LIN {X 0,Y 370.907,Z 638.749,A -85,B 0,C 180,E1 -12853.488,E2 -12853.488} C_VEL
LIN {X 0,Y 369.621,Z 646.813,A -85,B 0,C 180,E1 -12855.864,E2 -12855.864} C_VEL
LIN {X 0,Y 368.614,Z 653.844,A -85,B 0,C 180,E1 -12858.452,E2 -12858.452} C_VEL
LIN {X 0,Y 367.975,Z 659.585,A -85,B 0,C 180,E1 -12861.211,E2 -12861.211} C_VEL
LIN {X 0,Y 367.683,Z 663.304,A -85,B 0,C 180,E1 -12863.69,E2 -12863.69} C_VEL
LIN {X 0,Y 367.515,Z 665.39,A -85,B 0,C 180,E1 -12865.613,E2 -12865.613} C_VEL
LIN {X 0,Y 367.433,Z 666.778,A -85,B 0,C 180,E1 -12867.808,E2 -12867.808} C_VEL
LIN {X 0,Y 367.455,Z 667.313,A -85,B 0,C 180,E1 -12870,E2 -12870} C_VEL
LIN {X 0,Y 367.425,Z 666.872,A -85,B 0,C 180,E1 -12872.034,E2 -12872.034} C_VEL
LIN {X 0,Y 366.804,Z 666.517,A -85,B 0,C 180,E1 -12872.948,E2 -12872.948} C_VEL
LIN {X 0,Y 364.039,Z 665.625,A -85,B 0,C 180,E1 -12874.433,E2 -12874.433} C_VEL
LIN {X 0,Y 361.697,Z 664.56,A -85,B 0,C 180,E1 -12875.627,E2 -12875.627} C_VEL
LIN {X 0,Y 360.71,Z 663.504,A -85,B 0,C 180,E1 -12876.542,E2 -12876.542} C_VEL
LIN {X 0,Y 360.64,Z 663.097,A -85,B 0,C 180,E1 -12876.85,E2 -12876.85} C_VEL
LIN {X 0,Y 361.004,Z 658.926,A -85,B 0,C 180,E1 -12879.525,E2 -12879.525} C_VEL
LIN {X 0,Y 361.59,Z 654.287,A -85,B 0,C 180,E1 -12881.776,E2 -12881.776} C_VEL
LIN {X 0,Y 362.727,Z 646.801,A -85,B 0,C 180,E1 -12884.589,E2 -12884.589} C_VEL
LIN {X 0,Y 364.17,Z 638.314,A -85,B 0,C 180,E1 -12887.116,E2 -12887.116} C_VEL
LIN {X 0,Y 365.899,Z 628.97,A -85,B 0,C 180,E1 -12889.392,E2 -12889.392} C_VEL
LIN {X 0,Y 367.605,Z 619.716,A -85,B 0,C 180,E1 -12891.3,E2 -12891.3} C_VEL
LIN {X 0,Y 369.724,Z 608.71,A -85,B 0,C 180,E1 -12893.23,E2 -12893.23} C_VEL
LIN {X 0,Y 372.107,Z 596.049,A -85,B 0,C 180,E1 -12895.093,E2 -12895.093} C_VEL
LIN {X 0,Y 374.536,Z 582.365,A -85,B 0,C 180,E1 -12896.766,E2 -12896.766} C_VEL
LIN {X 0,Y 376.71,Z 569.237,A -85,B 0,C 180,E1 -12898.103,E2 -12898.103} C_VEL
LIN {X 0,Y 378.659,Z 555.105,A -85,B 0,C 180,E1 -12899.324,E2 -12899.324} C_VEL
LIN {X 0,Y 380.626,Z 540.226,A -85,B 0,C 180,E1 -12900.362,E2 -12900.362} C_VEL
LIN {X 0,Y 382.44,Z 523.413,A -85,B 0,C 180,E1 -12901.274,E2 -12901.274} C_VEL
LIN {X 0,Y 383.681,Z 507.284,A -85,B 0,C 180,E1 -12901.932,E2 -12901.932} C_VEL
LIN {X 0,Y 384.653,Z 490.648,A -85,B 0,C 180,E1 -12902.392,E2 -12902.392} C_VEL
LIN {X 0,Y 389.159,Z 339.278,A -85,B 0,C 180,E1 -12905.281,E2 -12905.281} C_VEL
LIN {X 0,Y 378.091,Z 317.354,A -85,B 0,C 180,E1 -12906.995,E2 -12906.995} C_VEL
LIN {X 0,Y 369.152,Z 301.874,A -85,B 0,C 180,E1 -12908.431,E2 -12908.431} C_VEL
LIN {X 0,Y 364.671,Z 294.925,A -85,B 0,C 180,E1 -12909.169,E2 -12909.169} C_VEL
LIN {X 0,Y 362.414,Z 291.756,A -85,B 0,C 180,E1 -12909.542,E2 -12909.542} C_VEL
LIN {X 0,Y 361.846,Z 289.718,A -85,B 0,C 180,E1 -12909.687,E2 -12909.687} C_VEL
LIN {X 0,Y 361.835,Z 289.718,A -85,B 0,C 180,E1 -12912.828,E2 -12912.828} C_VEL
LIN {X 0,Y 361.816,Z 289.719,A -85,B 0,C 180,E1 -12915.946,E2 -12915.946} C_VEL
LIN {X 0,Y 361.833,Z 289.715,A -85,B 0,C 180,E1 -12919.244,E2 -12919.244} C_VEL
LIN {X 0,Y 361.861,Z 289.71,A -85,B 0,C 180,E1 -12922.777,E2 -12922.777} C_VEL
LIN {X 0,Y 361.852,Z 289.721,A -85,B 0,C 180,E1 -12925.719,E2 -12925.719} C_VEL
LIN {X 0,Y 361.871,Z 289.722,A -85,B 0,C 180,E1 -12929.672,E2 -12929.672} C_VEL
LIN {X 0,Y 361.952,Z 289.699,A -85,B 0,C 180,E1 -12933.475,E2 -12933.475} C_VEL
LIN {X 0,Y 361.889,Z 289.7,A -85,B 0,C 180,E1 -12937.144,E2 -12937.144} C_VEL
LIN {X 0,Y 361.906,Z 289.717,A -85,B 0,C 180,E1 -12940.723,E2 -12940.723} C_VEL
LIN {X 0,Y 361.93,Z 289.693,A -85,B 0,C 180,E1 -12943.066,E2 -12943.066} C_VEL
LIN {X 0,Y 361.996,Z 289.703,A -85,B 0,C 180,E1 -12946.528,E2 -12946.528} C_VEL
LIN {X 0,Y 362.029,Z 289.677,A -85,B 0,C 180,E1 -12949.938,E2 -12949.938} C_VEL
LIN {X 0,Y 362.149,Z 289.678,A -85,B 0,C 180,E1 -12952.192,E2 -12952.192} C_VEL
LIN {X 0,Y 362.116,Z 289.69,A -85,B 0,C 180,E1 -12954.431,E2 -12954.431} C_VEL
LIN {X 0,Y 362.278,Z 289.647,A -85,B 0,C 180,E1 -12957.776,E2 -12957.776} C_VEL
LIN {X 0,Y 362.425,Z 289.65,A -85,B 0,C 180,E1 -12960,E2 -12960} C_VEL
LIN {X 0,Y 362.28,Z 289.662,A -85,B 0,C 180,E1 -12962.223,E2 -12962.223} C_VEL
LIN {X 0,Y 362.17,Z 289.682,A -85,B 0,C 180,E1 -12966.686,E2 -12966.686} C_VEL
LIN {X 0,Y 362.071,Z 289.684,A -85,B 0,C 180,E1 -12968.933,E2 -12968.933} C_VEL
LIN {X 0,Y 361.957,Z 289.702,A -85,B 0,C 180,E1 -12972.332,E2 -12972.332} C_VEL
LIN {X 0,Y 361.959,Z 289.709,A -85,B 0,C 180,E1 -12974.62,E2 -12974.62} C_VEL
LIN {X 0,Y 361.957,Z 289.707,A -85,B 0,C 180,E1 -12978.099,E2 -12978.099} C_VEL
LIN {X 0,Y 361.889,Z 289.717,A -85,B 0,C 180,E1 -12981.653,E2 -12981.653} C_VEL
LIN {X 0,Y 361.925,Z 289.718,A -85,B 0,C 180,E1 -12985.29,E2 -12985.29} C_VEL
LIN {X 0,Y 361.915,Z 289.716,A -85,B 0,C 180,E1 -12987.778,E2 -12987.778} C_VEL
LIN {X 0,Y 361.844,Z 289.731,A -85,B 0,C 180,E1 -12991.285,E2 -12991.285} C_VEL
LIN {X 0,Y 361.851,Z 289.729,A -85,B 0,C 180,E1 -12994.28,E2 -12994.28} C_VEL
LIN {X 0,Y 361.862,Z 289.728,A -85,B 0,C 180,E1 -12997.223,E2 -12997.223} C_VEL
LIN {X 0,Y 361.833,Z 289.733,A -85,B 0,C 180,E1 -13000.756,E2 -13000.756} C_VEL
LIN {X 0,Y 361.816,Z 289.734,A -85,B 0,C 180,E1 -13004.368,E2 -13004.368} C_VEL
LIN {X 0,Y 361.831,Z 289.732,A -85,B 0,C 180,E1 -13007.744,E2 -13007.744} C_VEL
LIN {X 0,Y 366.657,Z 302.939,A -85,B 0,C 180,E1 -13010.56,E2 -13010.56} C_VEL
LIN {X 0,Y 367.781,Z 306.002,A -85,B 0,C 180,E1 -13011.134,E2 -13011.134} C_VEL
LIN {X 0,Y 378.049,Z 324.644,A -85,B 0,C 180,E1 -13012.805,E2 -13012.805} C_VEL
LIN {X 0,Y 387.494,Z 344.135,A -85,B 0,C 180,E1 -13014.286,E2 -13014.286} C_VEL
LIN {X 0,Y 388.307,Z 346.732,A -85,B 0,C 180,E1 -13014.43,E2 -13014.43} C_VEL
LIN {X 0,Y 388.915,Z 352.418,A -85,B 0,C 180,E1 -13014.619,E2 -13014.619} C_VEL
LIN {X 0,Y 384.083,Z 512.924,A -85,B 0,C 180,E1 -13017.685,E2 -13017.685} C_VEL
LIN {X 0,Y 382.968,Z 528.887,A -85,B 0,C 180,E1 -13018.157,E2 -13018.157} C_VEL
LIN {X 0,Y 381.501,Z 544.325,A -85,B 0,C 180,E1 -13018.794,E2 -13018.794} C_VEL
LIN {X 0,Y 379.765,Z 559.811,A -85,B 0,C 180,E1 -13019.639,E2 -13019.639} C_VEL
LIN {X 0,Y 377.615,Z 575.779,A -85,B 0,C 180,E1 -13020.755,E2 -13020.755} C_VEL
LIN {X 0,Y 375.218,Z 591.049,A -85,B 0,C 180,E1 -13022.079,E2 -13022.079} C_VEL
LIN {X 0,Y 372.743,Z 605.042,A -85,B 0,C 180,E1 -13023.549,E2 -13023.549} C_VEL
LIN {X 0,Y 370.628,Z 617.005,A -85,B 0,C 180,E1 -13025.045,E2 -13025.045} C_VEL
LIN {X 0,Y 368.639,Z 628.246,A -85,B 0,C 180,E1 -13026.697,E2 -13026.697} C_VEL
LIN {X 0,Y 366.551,Z 639.457,A -85,B 0,C 180,E1 -13028.636,E2 -13028.636} C_VEL
LIN {X 0,Y 364.551,Z 650.326,A -85,B 0,C 180,E1 -13030.869,E2 -13030.869} C_VEL
LIN {X 0,Y 363.096,Z 659.472,A -85,B 0,C 180,E1 -13033.122,E2 -13033.122} C_VEL
LIN {X 0,Y 361.974,Z 667.139,A -85,B 0,C 180,E1 -13035.38,E2 -13035.38} C_VEL
LIN {X 0,Y 361.197,Z 673.403,A -85,B 0,C 180,E1 -13037.641,E2 -13037.641} C_VEL
LIN {X 0,Y 360.634,Z 678.538,A -85,B 0,C 180,E1 -13039.899,E2 -13039.899} C_VEL
LIN {X 0,Y 360.451,Z 682.536,A -85,B 0,C 180,E1 -13042.156,E2 -13042.156} C_VEL
LIN {X 0,Y 360.326,Z 685.494,A -85,B 0,C 180,E1 -13044.404,E2 -13044.404} C_VEL
LIN {X 0,Y 360.277,Z 687.443,A -85,B 0,C 180,E1 -13046.645,E2 -13046.645} C_VEL
LIN {X 0,Y 360.312,Z 688.409,A -85,B 0,C 180,E1 -13048.882,E2 -13048.882} C_VEL
LIN {X 0,Y 360.312,Z 688.408,A -85,B 0,C 180,E1 -13051.118,E2 -13051.118} C_VEL
LIN {X 0,Y 360.277,Z 687.435,A -85,B 0,C 180,E1 -13053.355,E2 -13053.355} C_VEL
LIN {X 0,Y 360.375,Z 685.105,A -85,B 0,C 180,E1 -13055.962,E2 -13055.962} C_VEL
LIN {X 0,Y 360.451,Z 682.522,A -85,B 0,C 180,E1 -13057.844,E2 -13057.844} C_VEL
LIN {X 0,Y 360.634,Z 678.523,A -85,B 0,C 180,E1 -13060.101,E2 -13060.101} C_VEL
LIN {X 0,Y 361.194,Z 673.38,A -85,B 0,C 180,E1 -13062.359,E2 -13062.359} C_VEL
LIN {X 0,Y 361.973,Z 667.108,A -85,B 0,C 180,E1 -13064.62,E2 -13064.62} C_VEL
LIN {X 0,Y 363.295,Z 658.416,A -85,B 0,C 180,E1 -13067.158,E2 -13067.158} C_VEL
LIN {X 0,Y 364.819,Z 649.165,A -85,B 0,C 180,E1 -13069.379,E2 -13069.379} C_VEL
LIN {X 0,Y 366.566,Z 639.399,A -85,B 0,C 180,E1 -13071.363,E2 -13071.363} C_VEL
LIN {X 0,Y 368.709,Z 628.173,A -85,B 0,C 180,E1 -13073.298,E2 -13073.298} C_VEL
LIN {X 0,Y 370.837,Z 615.941,A -85,B 0,C 180,E1 -13075.09,E2 -13075.09} C_VEL
LIN {X 0,Y 373.179,Z 602.583,A -85,B 0,C 180,E1 -13076.72,E2 -13076.72} C_VEL
LIN {X 0,Y 375.461,Z 589.361,A -85,B 0,C 180,E1 -13078.067,E2 -13078.067} C_VEL
LIN {X 0,Y 377.374,Z 577.294,A -85,B 0,C 180,E1 -13079.113,E2 -13079.113} C_VEL
LIN {X 0,Y 379.367,Z 562.609,A -85,B 0,C 180,E1 -13080.166,E2 -13080.166} C_VEL
LIN {X 0,Y 381.26,Z 546.692,A -85,B 0,C 180,E1 -13081.074,E2 -13081.074} C_VEL
LIN {X 0,Y 382.736,Z 531.3,A -85,B 0,C 180,E1 -13081.749,E2 -13081.749} C_VEL
LIN {X 0,Y 384.045,Z 514.1,A -85,B 0,C 180,E1 -13082.273,E2 -13082.273} C_VEL
LIN {X 0,Y 388.906,Z 351.926,A -85,B 0,C 180,E1 -13085.377,E2 -13085.377} C_VEL
LIN {X 0,Y 388.013,Z 345.342,A -85,B 0,C 180,E1 -13085.616,E2 -13085.616} C_VEL
LIN {X 0,Y 379.342,Z 327.267,A -85,B 0,C 180,E1 -13086.969,E2 -13086.969} C_VEL
LIN {X 0,Y 369.961,Z 309.878,A -85,B 0,C 180,E1 -13088.481,E2 -13088.481} C_VEL
LIN {X 0,Y 367.493,Z 305.339,A -85,B 0,C 180,E1 -13088.93,E2 -13088.93} C_VEL
LIN {X 0,Y 363.709,Z 294.968,A -85,B 0,C 180,E1 -13091.097,E2 -13091.097} C_VEL
LIN {X 0,Y 361.832,Z 289.724,A -85,B 0,C 180,E1 -13092.271,E2 -13092.271} C_VEL
LIN {X 0,Y 361.833,Z 289.72,A -85,B 0,C 180,E1 -13095.944,E2 -13095.944} C_VEL
LIN {X 0,Y 361.833,Z 289.724,A -85,B 0,C 180,E1 -13099.245,E2 -13099.245} C_VEL
LIN {X 0,Y 361.861,Z 289.715,A -85,B 0,C 180,E1 -13102.777,E2 -13102.777} C_VEL
LIN {X 0,Y 361.852,Z 289.721,A -85,B 0,C 180,E1 -13105.72,E2 -13105.72} C_VEL
LIN {X 0,Y 361.872,Z 289.716,A -85,B 0,C 180,E1 -13109.672,E2 -13109.672} C_VEL
LIN {X 0,Y 361.952,Z 289.711,A -85,B 0,C 180,E1 -13113.475,E2 -13113.475} C_VEL
LIN {X 0,Y 361.89,Z 289.721,A -85,B 0,C 180,E1 -13117.145,E2 -13117.145} C_VEL
LIN {X 0,Y 361.909,Z 289.693,A -85,B 0,C 180,E1 -13120.724,E2 -13120.724} C_VEL
LIN {X 0,Y 361.931,Z 289.716,A -85,B 0,C 180,E1 -13123.066,E2 -13123.066} C_VEL
LIN {X 0,Y 361.996,Z 289.677,A -85,B 0,C 180,E1 -13126.528,E2 -13126.528} C_VEL
LIN {X 0,Y 362.029,Z 289.701,A -85,B 0,C 180,E1 -13129.938,E2 -13129.938} C_VEL
LIN {X 0,Y 362.161,Z 289.655,A -85,B 0,C 180,E1 -13133.314,E2 -13133.314} C_VEL
LIN {X 0,Y 362.281,Z 289.668,A -85,B 0,C 180,E1 -13137.777,E2 -13137.777} C_VEL
LIN {X 0,Y 362.424,Z 289.626,A -85,B 0,C 180,E1 -13140,E2 -13140} C_VEL
LIN {X 0,Y 362.279,Z 289.653,A -85,B 0,C 180,E1 -13142.224,E2 -13142.224} C_VEL
LIN {X 0,Y 362.161,Z 289.665,A -85,B 0,C 180,E1 -13146.687,E2 -13146.687} C_VEL
LIN {X 0,Y 362.03,Z 289.692,A -85,B 0,C 180,E1 -13150.062,E2 -13150.062} C_VEL
LIN {X 0,Y 361.996,Z 289.69,A -85,B 0,C 180,E1 -13153.899,E2 -13153.899} C_VEL
LIN {X 0,Y 361.966,Z 289.707,A -85,B 0,C 180,E1 -13157.939,E2 -13157.939} C_VEL
LIN {X 0,Y 361.882,Z 289.692,A -85,B 0,C 180,E1 -13161.654,E2 -13161.654} C_VEL
LIN {X 0,Y 361.927,Z 289.714,A -85,B 0,C 180,E1 -13165.29,E2 -13165.29} C_VEL
LIN {X 0,Y 361.907,Z 289.692,A -85,B 0,C 180,E1 -13167.779,E2 -13167.779} C_VEL
LIN {X 0,Y 361.836,Z 289.72,A -85,B 0,C 180,E1 -13171.63,E2 -13171.63} C_VEL
LIN {X 0,Y 361.873,Z 289.72,A -85,B 0,C 180,E1 -13175.345,E2 -13175.345} C_VEL
LIN {X 0,Y 361.867,Z 289.707,A -85,B 0,C 180,E1 -13179.027,E2 -13179.027} C_VEL
LIN {X 0,Y 361.835,Z 289.711,A -85,B 0,C 180,E1 -13182.829,E2 -13182.829} C_VEL
LIN {X 0,Y 361.816,Z 289.715,A -85,B 0,C 180,E1 -13185.947,E2 -13185.947} C_VEL
LIN {X 0,Y 361.835,Z 289.727,A -85,B 0,C 180,E1 -13189.245,E2 -13189.245} C_VEL
LIN {X 0,Y 361.839,Z 289.728,A -85,B 0,C 180,E1 -13190.441,E2 -13190.441} C_VEL
LIN {X 0,Y 362.896,Z 292.623,A -85,B 0,C 180,E1 -13190.657,E2 -13190.657} C_VEL
LIN {X 0,Y 364.71,Z 294.95,A -85,B 0,C 180,E1 -13190.95,E2 -13190.95} C_VEL
LIN {X 0,Y 372.447,Z 307.404,A -85,B 0,C 180,E1 -13192.216,E2 -13192.216} C_VEL
LIN {X 0,Y 380.406,Z 321.844,A -85,B 0,C 180,E1 -13193.481,E2 -13193.481} C_VEL
LIN {X 0,Y 389.033,Z 339.103,A -85,B 0,C 180,E1 -13194.808,E2 -13194.808} C_VEL
LIN {X 0,Y 384.556,Z 492.624,A -85,B 0,C 180,E1 -13197.755,E2 -13197.755} C_VEL
LIN {X 0,Y 383.59,Z 508.462,A -85,B 0,C 180,E1 -13198.214,E2 -13198.214} C_VEL
LIN {X 0,Y 382.299,Z 524.246,A -85,B 0,C 180,E1 -13198.867,E2 -13198.867} C_VEL
LIN {X 0,Y 380.624,Z 539.824,A -85,B 0,C 180,E1 -13199.715,E2 -13199.715} C_VEL
LIN {X 0,Y 378.562,Z 555.625,A -85,B 0,C 180,E1 -13200.818,E2 -13200.818} C_VEL
LIN {X 0,Y 376.568,Z 569.681,A -85,B 0,C 180,E1 -13202.036,E2 -13202.036} C_VEL
LIN {X 0,Y 374.451,Z 582.728,A -85,B 0,C 180,E1 -13203.378,E2 -13203.378} C_VEL
LIN {X 0,Y 372.228,Z 595.02,A -85,B 0,C 180,E1 -13204.871,E2 -13204.871} C_VEL
LIN {X 0,Y 370.133,Z 606.325,A -85,B 0,C 180,E1 -13206.501,E2 -13206.501} C_VEL
LIN {X 0,Y 367.956,Z 617.73,A -85,B 0,C 180,E1 -13208.428,E2 -13208.428} C_VEL
LIN {X 0,Y 366.253,Z 626.909,A -85,B 0,C 180,E1 -13210.251,E2 -13210.251} C_VEL
LIN {X 0,Y 364.597,Z 635.754,A -85,B 0,C 180,E1 -13212.326,E2 -13212.326} C_VEL
LIN {X 0,Y 363.367,Z 642.912,A -85,B 0,C 180,E1 -13214.29,E2 -13214.29} C_VEL
LIN {X 0,Y 362.22,Z 649.717,A -85,B 0,C 180,E1 -13216.536,E2 -13216.536} C_VEL
LIN {X 0,Y 361.389,Z 655.303,A -85,B 0,C 180,E1 -13218.786,E2 -13218.786} C_VEL
LIN {X 0,Y 360.944,Z 659.793,A -85,B 0,C 180,E1 -13221.039,E2 -13221.039} C_VEL
LIN {X 0,Y 360.587,Z 663.718,A -85,B 0,C 180,E1 -13223.727,E2 -13223.727} C_VEL
LIN {X 0,Y 360.449,Z 665.597,A -85,B 0,C 180,E1 -13225.527,E2 -13225.527} C_VEL
LIN {X 0,Y 360.334,Z 666.986,A -85,B 0,C 180,E1 -13227.764,E2 -13227.764} C_VEL
LIN {X 0,Y 360.359,Z 667.52,A -85,B 0,C 180,E1 -13230,E2 -13230} C_VEL
LIN {X 0,Y 360.334,Z 667.029,A -85,B 0,C 180,E1 -13232.236,E2 -13232.236} C_VEL
LIN {X 0,Y 360.448,Z 665.682,A -85,B 0,C 180,E1 -13234.473,E2 -13234.473} C_VEL
LIN {X 0,Y 360.64,Z 663.097,A -85,B 0,C 180,E1 -13236.85,E2 -13236.85} C_VEL
LIN {X 0,Y 360.022,Z 661.911,A -85,B 0,C 180,E1 -13237.763,E2 -13237.763} C_VEL
LIN {X 0,Y 357.323,Z 659.723,A -85,B 0,C 180,E1 -13239.249,E2 -13239.249} C_VEL
LIN {X 0,Y 354.789,Z 657.157,A -85,B 0,C 180,E1 -13240.741,E2 -13240.741} C_VEL
LIN {X 0,Y 354.443,Z 655.273,A -85,B 0,C 180,E1 -13241.65,E2 -13241.65} C_VEL
LIN {X 0,Y 355.247,Z 650.204,A -85,B 0,C 180,E1 -13243.733,E2 -13243.733} C_VEL
LIN {X 0,Y 356.422,Z 643.435,A -85,B 0,C 180,E1 -13246.025,E2 -13246.025} C_VEL
LIN {X 0,Y 357.944,Z 635.243,A -85,B 0,C 180,E1 -13248.309,E2 -13248.309} C_VEL
LIN {X 0,Y 359.824,Z 625.486,A -85,B 0,C 180,E1 -13250.583,E2 -13250.583} C_VEL
LIN {X 0,Y 361.853,Z 615.447,A -85,B 0,C 180,E1 -13252.556,E2 -13252.556} C_VEL
LIN {X 0,Y 364.176,Z 603.608,A -85,B 0,C 180,E1 -13254.514,E2 -13254.514} C_VEL
LIN {X 0,Y 366.713,Z 590.572,A -85,B 0,C 180,E1 -13256.307,E2 -13256.307} C_VEL
LIN {X 0,Y 368.98,Z 577.552,A -85,B 0,C 180,E1 -13257.817,E2 -13257.817} C_VEL
LIN {X 0,Y 371.334,Z 563.556,A -85,B 0,C 180,E1 -13259.166,E2 -13259.166} C_VEL
LIN {X 0,Y 373.238,Z 550.201,A -85,B 0,C 180,E1 -13260.244,E2 -13260.244} C_VEL
LIN {X 0,Y 375.08,Z 535.938,A -85,B 0,C 180,E1 -13261.172,E2 -13261.172} C_VEL
LIN {X 0,Y 376.727,Z 519.187,A -85,B 0,C 180,E1 -13262.04,E2 -13262.04} C_VEL
LIN {X 0,Y 378.038,Z 503.614,A -85,B 0,C 180,E1 -13262.624,E2 -13262.624} C_VEL
LIN {X 0,Y 378.868,Z 486.851,A -85,B 0,C 180,E1 -13263.053,E2 -13263.053} C_VEL
LIN {X 0,Y 383.292,Z 341.409,A -85,B 0,C 180,E1 -13265.859,E2 -13265.859} C_VEL
LIN {X 0,Y 372.607,Z 320.441,A -85,B 0,C 180,E1 -13267.563,E2 -13267.563} C_VEL
LIN {X 0,Y 364.726,Z 306.671,A -85,B 0,C 180,E1 -13268.869,E2 -13268.869} C_VEL
LIN {X 0,Y 358.95,Z 298.084,A -85,B 0,C 180,E1 -13269.841,E2 -13269.841} C_VEL
LIN {X 0,Y 357.037,Z 294.944,A -85,B 0,C 180,E1 -13270.18,E2 -13270.18} C_VEL
LIN {X 0,Y 355.371,Z 292.659,A -85,B 0,C 180,E1 -13270.468,E2 -13270.468} C_VEL
LIN {X 0,Y 354.794,Z 290.6,A -85,B 0,C 180,E1 -13270.637,E2 -13270.637} C_VEL
LIN {X 0,Y 354.766,Z 290.608,A -85,B 0,C 180,E1 -13273.896,E2 -13273.896} C_VEL
LIN {X 0,Y 354.793,Z 290.601,A -85,B 0,C 180,E1 -13277.662,E2 -13277.662} C_VEL
LIN {X 0,Y 354.814,Z 290.6,A -85,B 0,C 180,E1 -13280.666,E2 -13280.666} C_VEL
LIN {X 0,Y 354.82,Z 290.596,A -85,B 0,C 180,E1 -13284.3,E2 -13284.3} C_VEL
LIN {X 0,Y 354.785,Z 290.588,A -85,B 0,C 180,E1 -13287.666,E2 -13287.666} C_VEL
LIN {X 0,Y 354.844,Z 290.58,A -85,B 0,C 180,E1 -13291.618,E2 -13291.618} C_VEL
LIN {X 0,Y 354.897,Z 290.587,A -85,B 0,C 180,E1 -13294.172,E2 -13294.172} C_VEL
LIN {X 0,Y 354.833,Z 290.574,A -85,B 0,C 180,E1 -13297.894,E2 -13297.894} C_VEL
LIN {X 0,Y 354.92,Z 290.582,A -85,B 0,C 180,E1 -13301.891,E2 -13301.891} C_VEL
LIN {X 0,Y 354.941,Z 290.58,A -85,B 0,C 180,E1 -13305.981,E2 -13305.981} C_VEL
LIN {X 0,Y 354.975,Z 290.557,A -85,B 0,C 180,E1 -13309.736,E2 -13309.736} C_VEL
LIN {X 0,Y 355.112,Z 290.552,A -85,B 0,C 180,E1 -13312.037,E2 -13312.037} C_VEL
LIN {X 0,Y 355.09,Z 290.565,A -85,B 0,C 180,E1 -13314.321,E2 -13314.321} C_VEL
LIN {X 0,Y 355.241,Z 290.522,A -85,B 0,C 180,E1 -13317.732,E2 -13317.732} C_VEL
LIN {X 0,Y 355.395,Z 290.526,A -85,B 0,C 180,E1 -13320,E2 -13320} C_VEL
LIN {X 0,Y 355.243,Z 290.536,A -85,B 0,C 180,E1 -13322.267,E2 -13322.267} C_VEL
LIN {X 0,Y 355.136,Z 290.559,A -85,B 0,C 180,E1 -13326.819,E2 -13326.819} C_VEL
LIN {X 0,Y 355.013,Z 290.561,A -85,B 0,C 180,E1 -13329.112,E2 -13329.112} C_VEL
LIN {X 0,Y 354.918,Z 290.58,A -85,B 0,C 180,E1 -13332.581,E2 -13332.581} C_VEL
LIN {X 0,Y 354.887,Z 290.589,A -85,B 0,C 180,E1 -13336.096,E2 -13336.096} C_VEL
LIN {X 0,Y 354.904,Z 290.585,A -85,B 0,C 180,E1 -13338.472,E2 -13338.472} C_VEL
LIN {X 0,Y 354.832,Z 290.597,A -85,B 0,C 180,E1 -13342.106,E2 -13342.106} C_VEL
LIN {X 0,Y 354.897,Z 290.593,A -85,B 0,C 180,E1 -13345.827,E2 -13345.827} C_VEL
LIN {X 0,Y 354.851,Z 290.596,A -85,B 0,C 180,E1 -13349.679,E2 -13349.679} C_VEL
LIN {X 0,Y 354.803,Z 290.606,A -85,B 0,C 180,E1 -13353.702,E2 -13353.702} C_VEL
LIN {X 0,Y 354.796,Z 290.606,A -85,B 0,C 180,E1 -13356.459,E2 -13356.459} C_VEL
LIN {X 0,Y 354.821,Z 290.605,A -85,B 0,C 180,E1 -13359.424,E2 -13359.424} C_VEL
LIN {X 0,Y 354.785,Z 290.61,A -85,B 0,C 180,E1 -13362.867,E2 -13362.867} C_VEL
LIN {X 0,Y 354.799,Z 290.69,A -85,B 0,C 180,E1 -13366.918,E2 -13366.918} C_VEL
LIN {X 0,Y 359.992,Z 304.716,A -85,B 0,C 180,E1 -13370.018,E2 -13370.018} C_VEL
LIN {X 0,Y 360.489,Z 305.861,A -85,B 0,C 180,E1 -13370.196,E2 -13370.196} C_VEL
LIN {X 0,Y 370.78,Z 324.284,A -85,B 0,C 180,E1 -13371.945,E2 -13371.945} C_VEL
LIN {X 0,Y 379.91,Z 342.544,A -85,B 0,C 180,E1 -13373.429,E2 -13373.429} C_VEL
LIN {X 0,Y 382.62,Z 348.545,A -85,B 0,C 180,E1 -13373.864,E2 -13373.864} C_VEL
LIN {X 0,Y 383.121,Z 353.621,A -85,B 0,C 180,E1 -13374.033,E2 -13374.033} C_VEL
LIN {X 0,Y 378.075,Z 513.451,A -85,B 0,C 180,E1 -13377.126,E2 -13377.126} C_VEL
LIN {X 0,Y 376.874,Z 529.607,A -85,B 0,C 180,E1 -13377.619,E2 -13377.619} C_VEL
LIN {X 0,Y 375.269,Z 545.427,A -85,B 0,C 180,E1 -13378.295,E2 -13378.295} C_VEL
LIN {X 0,Y 373.489,Z 560.605,A -85,B 0,C 180,E1 -13379.152,E2 -13379.152} C_VEL
LIN {X 0,Y 371.387,Z 575.575,A -85,B 0,C 180,E1 -13380.215,E2 -13380.215} C_VEL
LIN {X 0,Y 368.906,Z 590.844,A -85,B 0,C 180,E1 -13381.558,E2 -13381.558} C_VEL
LIN {X 0,Y 366.354,Z 604.837,A -85,B 0,C 180,E1 -13383.05,E2 -13383.05} C_VEL
LIN {X 0,Y 364.069,Z 616.796,A -85,B 0,C 180,E1 -13384.564,E2 -13384.564} C_VEL
LIN {X 0,Y 362.036,Z 628.038,A -85,B 0,C 180,E1 -13386.246,E2 -13386.246} C_VEL
LIN {X 0,Y 359.839,Z 639.248,A -85,B 0,C 180,E1 -13388.218,E2 -13388.218} C_VEL
LIN {X 0,Y 357.782,Z 650.118,A -85,B 0,C 180,E1 -13390.492,E2 -13390.492} C_VEL
LIN {X 0,Y 356.204,Z 659.263,A -85,B 0,C 180,E1 -13392.785,E2 -13392.785} C_VEL
LIN {X 0,Y 355.007,Z 666.93,A -85,B 0,C 180,E1 -13395.087,E2 -13395.087} C_VEL
LIN {X 0,Y 354.191,Z 673.194,A -85,B 0,C 180,E1 -13397.393,E2 -13397.393} C_VEL
LIN {X 0,Y 353.578,Z 678.329,A -85,B 0,C 180,E1 -13399.695,E2 -13399.695} C_VEL
LIN {X 0,Y 353.362,Z 682.328,A -85,B 0,C 180,E1 -13401.997,E2 -13401.997} C_VEL
LIN {X 0,Y 353.259,Z 685.287,A -85,B 0,C 180,E1 -13404.291,E2 -13404.291} C_VEL
LIN {X 0,Y 353.197,Z 687.236,A -85,B 0,C 180,E1 -13406.578,E2 -13406.578} C_VEL
LIN {X 0,Y 353.212,Z 688.202,A -85,B 0,C 180,E1 -13408.86,E2 -13408.86} C_VEL
LIN {X 0,Y 353.212,Z 688.2,A -85,B 0,C 180,E1 -13411.14,E2 -13411.14} C_VEL
LIN {X 0,Y 353.197,Z 687.228,A -85,B 0,C 180,E1 -13413.422,E2 -13413.422} C_VEL
LIN {X 0,Y 353.275,Z 685.077,A -85,B 0,C 180,E1 -13415.908,E2 -13415.908} C_VEL
LIN {X 0,Y 353.362,Z 682.313,A -85,B 0,C 180,E1 -13418.003,E2 -13418.003} C_VEL
LIN {X 0,Y 353.578,Z 678.313,A -85,B 0,C 180,E1 -13420.305,E2 -13420.305} C_VEL
LIN {X 0,Y 354.188,Z 673.17,A -85,B 0,C 180,E1 -13422.607,E2 -13422.607} C_VEL
LIN {X 0,Y 355.006,Z 666.896,A -85,B 0,C 180,E1 -13424.913,E2 -13424.913} C_VEL
LIN {X 0,Y 356.431,Z 658.205,A -85,B 0,C 180,E1 -13427.499,E2 -13427.499} C_VEL
LIN {X 0,Y 358.026,Z 648.827,A -85,B 0,C 180,E1 -13429.792,E2 -13429.792} C_VEL
LIN {X 0,Y 359.848,Z 639.186,A -85,B 0,C 180,E1 -13431.782,E2 -13431.782} C_VEL
LIN {X 0,Y 362.085,Z 627.96,A -85,B 0,C 180,E1 -13433.75,E2 -13433.75} C_VEL
LIN {X 0,Y 364.317,Z 615.728,A -85,B 0,C 180,E1 -13435.571,E2 -13435.571} C_VEL
LIN {X 0,Y 366.789,Z 602.371,A -85,B 0,C 180,E1 -13437.224,E2 -13437.224} C_VEL
LIN {X 0,Y 369.299,Z 588.05,A -85,B 0,C 180,E1 -13438.697,E2 -13438.697} C_VEL
LIN {X 0,Y 371.621,Z 573.626,A -85,B 0,C 180,E1 -13439.92,E2 -13439.92} C_VEL
LIN {X 0,Y 373.773,Z 558.304,A -85,B 0,C 180,E1 -13440.979,E2 -13440.979} C_VEL
LIN {X 0,Y 375.571,Z 542.568,A -85,B 0,C 180,E1 -13441.834,E2 -13441.834} C_VEL
LIN {X 0,Y 377.076,Z 526.494,A -85,B 0,C 180,E1 -13442.48,E2 -13442.48} C_VEL
LIN {X 0,Y 378.261,Z 510.347,A -85,B 0,C 180,E1 -13442.922,E2 -13442.922} C_VEL
LIN {X 0,Y 383.037,Z 351.609,A -85,B 0,C 180,E1 -13446.004,E2 -13446.004} C_VEL
LIN {X 0,Y 382.42,Z 348.085,A -85,B 0,C 180,E1 -13446.151,E2 -13446.151} C_VEL
LIN {X 0,Y 373.879,Z 330.341,A -85,B 0,C 180,E1 -13447.524,E2 -13447.524} C_VEL
LIN {X 0,Y 365.281,Z 314.342,A -85,B 0,C 180,E1 -13448.952,E2 -13448.952} C_VEL
LIN {X 0,Y 360.178,Z 305.201,A -85,B 0,C 180,E1 -13449.854,E2 -13449.854} C_VEL
LIN {X 0,Y 355.516,Z 292.944,A -85,B 0,C 180,E1 -13452.556,E2 -13452.556} C_VEL
LIN {X 0,Y 354.782,Z 290.602,A -85,B 0,C 180,E1 -13453.079,E2 -13453.079} C_VEL
LIN {X 0,Y 354.778,Z 290.598,A -85,B 0,C 180,E1 -13456.106,E2 -13456.106} C_VEL
LIN {X 0,Y 354.785,Z 290.601,A -85,B 0,C 180,E1 -13459.179,E2 -13459.179} C_VEL
LIN {X 0,Y 354.804,Z 290.594,A -85,B 0,C 180,E1 -13462.403,E2 -13462.403} C_VEL
LIN {X 0,Y 354.809,Z 290.594,A -85,B 0,C 180,E1 -13464.941,E2 -13464.941} C_VEL
LIN {X 0,Y 354.791,Z 290.6,A -85,B 0,C 180,E1 -13468.405,E2 -13468.405} C_VEL
LIN {X 0,Y 354.849,Z 290.595,A -85,B 0,C 180,E1 -13471.619,E2 -13471.619} C_VEL
LIN {X 0,Y 354.897,Z 290.589,A -85,B 0,C 180,E1 -13474.173,E2 -13474.173} C_VEL
LIN {X 0,Y 354.834,Z 290.593,A -85,B 0,C 180,E1 -13477.894,E2 -13477.894} C_VEL
LIN {X 0,Y 354.92,Z 290.581,A -85,B 0,C 180,E1 -13481.892,E2 -13481.892} C_VEL
LIN {X 0,Y 354.94,Z 290.557,A -85,B 0,C 180,E1 -13485.981,E2 -13485.981} C_VEL
LIN {X 0,Y 354.976,Z 290.58,A -85,B 0,C 180,E1 -13489.736,E2 -13489.736} C_VEL
LIN {X 0,Y 355.124,Z 290.531,A -85,B 0,C 180,E1 -13493.181,E2 -13493.181} C_VEL
LIN {X 0,Y 355.244,Z 290.544,A -85,B 0,C 180,E1 -13497.733,E2 -13497.733} C_VEL
LIN {X 0,Y 355.373,Z 290.503,A -85,B 0,C 180,E1 -13500,E2 -13500} C_VEL
LIN {X 0,Y 355.242,Z 290.529,A -85,B 0,C 180,E1 -13502.268,E2 -13502.268} C_VEL
LIN {X 0,Y 355.124,Z 290.539,A -85,B 0,C 180,E1 -13506.82,E2 -13506.82} C_VEL
LIN {X 0,Y 354.976,Z 290.571,A -85,B 0,C 180,E1 -13510.264,E2 -13510.264} C_VEL
LIN {X 0,Y 354.941,Z 290.565,A -85,B 0,C 180,E1 -13514.019,E2 -13514.019} C_VEL
LIN {X 0,Y 354.921,Z 290.585,A -85,B 0,C 180,E1 -13518.109,E2 -13518.109} C_VEL
LIN {X 0,Y 354.829,Z 290.57,A -85,B 0,C 180,E1 -13522.107,E2 -13522.107} C_VEL
LIN {X 0,Y 354.898,Z 290.587,A -85,B 0,C 180,E1 -13525.828,E2 -13525.828} C_VEL
LIN {X 0,Y 354.845,Z 290.593,A -85,B 0,C 180,E1 -13529.68,E2 -13529.68} C_VEL
LIN {X 0,Y 354.805,Z 290.599,A -85,B 0,C 180,E1 -13533.702,E2 -13533.702} C_VEL
LIN {X 0,Y 354.797,Z 290.597,A -85,B 0,C 180,E1 -13536.46,E2 -13536.46} C_VEL
LIN {X 0,Y 354.823,Z 290.59,A -85,B 0,C 180,E1 -13539.424,E2 -13539.424} C_VEL
LIN {X 0,Y 354.787,Z 290.589,A -85,B 0,C 180,E1 -13542.867,E2 -13542.867} C_VEL
LIN {X 0,Y 354.765,Z 290.593,A -85,B 0,C 180,E1 -13546.104,E2 -13546.104} C_VEL
LIN {X 0,Y 354.789,Z 290.604,A -85,B 0,C 180,E1 -13549.503,E2 -13549.503} C_VEL
LIN {X 0,Y 355.805,Z 293.453,A -85,B 0,C 180,E1 -13549.728,E2 -13549.728} C_VEL
LIN {X 0,Y 357.773,Z 295.999,A -85,B 0,C 180,E1 -13550.063,E2 -13550.063} C_VEL
LIN {X 0,Y 359.906,Z 299.245,A -85,B 0,C 180,E1 -13550.431,E2 -13550.431} C_VEL
LIN {X 0,Y 367.872,Z 311.995,A -85,B 0,C 180,E1 -13551.769,E2 -13551.769} C_VEL
LIN {X 0,Y 375.815,Z 326.553,A -85,B 0,C 180,E1 -13553.068,E2 -13553.068} C_VEL
LIN {X 0,Y 383.232,Z 341.44,A -85,B 0,C 180,E1 -13554.242,E2 -13554.242} C_VEL
LIN {X 0,Y 378.542,Z 494.115,A -85,B 0,C 180,E1 -13557.212,E2 -13557.212} C_VEL
LIN {X 0,Y 377.432,Z 510.511,A -85,B 0,C 180,E1 -13557.712,E2 -13557.712} C_VEL
LIN {X 0,Y 375.997,Z 527.053,A -85,B 0,C 180,E1 -13558.442,E2 -13558.442} C_VEL
LIN {X 0,Y 374.126,Z 543.058,A -85,B 0,C 180,E1 -13559.367,E2 -13559.367} C_VEL
LIN {X 0,Y 372.049,Z 558.335,A -85,B 0,C 180,E1 -13560.486,E2 -13560.486} C_VEL
LIN {X 0,Y 369.818,Z 572.735,A -85,B 0,C 180,E1 -13561.789,E2 -13561.789} C_VEL
LIN {X 0,Y 367.401,Z 586.442,A -85,B 0,C 180,E1 -13563.287,E2 -13563.287} C_VEL
LIN {X 0,Y 365.031,Z 599.117,A -85,B 0,C 180,E1 -13564.94,E2 -13564.94} C_VEL
LIN {X 0,Y 362.944,Z 610.043,A -85,B 0,C 180,E1 -13566.612,E2 -13566.612} C_VEL
LIN {X 0,Y 360.701,Z 620.889,A -85,B 0,C 180,E1 -13568.572,E2 -13568.572} C_VEL
LIN {X 0,Y 358.937,Z 630.155,A -85,B 0,C 180,E1 -13570.558,E2 -13570.558} C_VEL
LIN {X 0,Y 357.168,Z 639.172,A -85,B 0,C 180,E1 -13572.833,E2 -13572.833} C_VEL
LIN {X 0,Y 355.864,Z 646.7,A -85,B 0,C 180,E1 -13575.123,E2 -13575.123} C_VEL
LIN {X 0,Y 354.619,Z 654.264,A -85,B 0,C 180,E1 -13577.989,E2 -13577.989} C_VEL
LIN {X 0,Y 353.883,Z 660.003,A -85,B 0,C 180,E1 -13580.858,E2 -13580.858} C_VEL
LIN {X 0,Y 353.501,Z 664.112,A -85,B 0,C 180,E1 -13583.75,E2 -13583.75} C_VEL
LIN {X 0,Y 353.362,Z 665.805,A -85,B 0,C 180,E1 -13585.437,E2 -13585.437} C_VEL
LIN {X 0,Y 353.238,Z 667.193,A -85,B 0,C 180,E1 -13587.719,E2 -13587.719} C_VEL
LIN {X 0,Y 353.262,Z 667.727,A -85,B 0,C 180,E1 -13590,E2 -13590} C_VEL
LIN {X 0,Y 353.238,Z 667.236,A -85,B 0,C 180,E1 -13592.28,E2 -13592.28} C_VEL
LIN {X 0,Y 353.362,Z 665.889,A -85,B 0,C 180,E1 -13594.563,E2 -13594.563} C_VEL
LIN {X 0,Y 353.577,Z 663.464,A -85,B 0,C 180,E1 -13596.868,E2 -13596.868} C_VEL
LIN {X 0,Y 353.872,Z 660.181,A -85,B 0,C 180,E1 -13599.142,E2 -13599.142} C_VEL
LIN {X 0,Y 354.443,Z 655.273,A -85,B 0,C 180,E1 -13601.65,E2 -13601.65} C_VEL
LIN {X 0,Y 354.138,Z 653.332,A -85,B 0,C 180,E1 -13602.551,E2 -13602.551} C_VEL
LIN {X 0,Y 351.877,Z 650.023,A -85,B 0,C 180,E1 -13604.025,E2 -13604.025} C_VEL
LIN {X 0,Y 349.702,Z 646.266,A -85,B 0,C 180,E1 -13605.488,E2 -13605.488} C_VEL
LIN {X 0,Y 349.539,Z 643.62,A -85,B 0,C 180,E1 -13606.356,E2 -13606.356} C_VEL
LIN {X 0,Y 351.155,Z 635.45,A -85,B 0,C 180,E1 -13608.676,E2 -13608.676} C_VEL
LIN {X 0,Y 353.122,Z 625.693,A -85,B 0,C 180,E1 -13610.992,E2 -13610.992} C_VEL
LIN {X 0,Y 355.255,Z 615.653,A -85,B 0,C 180,E1 -13612.999,E2 -13612.999} C_VEL
LIN {X 0,Y 357.637,Z 604.059,A -85,B 0,C 180,E1 -13614.949,E2 -13614.949} C_VEL
LIN {X 0,Y 360.119,Z 591.839,A -85,B 0,C 180,E1 -13616.67,E2 -13616.67} C_VEL
LIN {X 0,Y 362.711,Z 577.755,A -85,B 0,C 180,E1 -13618.341,E2 -13618.341} C_VEL
LIN {X 0,Y 365.117,Z 563.798,A -85,B 0,C 180,E1 -13619.708,E2 -13619.708} C_VEL
LIN {X 0,Y 367.076,Z 550.75,A -85,B 0,C 180,E1 -13620.775,E2 -13620.775} C_VEL
LIN {X 0,Y 369.024,Z 536.137,A -85,B 0,C 180,E1 -13621.743,E2 -13621.743} C_VEL
LIN {X 0,Y 370.736,Z 519.383,A -85,B 0,C 180,E1 -13622.621,E2 -13622.621} C_VEL
LIN {X 0,Y 372.096,Z 503.805,A -85,B 0,C 180,E1 -13623.212,E2 -13623.212} C_VEL
LIN {X 0,Y 372.946,Z 486.848,A -85,B 0,C 180,E1 -13623.652,E2 -13623.652} C_VEL
LIN {X 0,Y 377.51,Z 343.742,A -85,B 0,C 180,E1 -13626.446,E2 -13626.446} C_VEL
LIN {X 0,Y 367.768,Z 324.625,A -85,B 0,C 180,E1 -13628.047,E2 -13628.047} C_VEL
LIN {X 0,Y 360.354,Z 311.572,A -85,B 0,C 180,E1 -13629.311,E2 -13629.311} C_VEL
LIN {X 0,Y 352.489,Z 299.627,A -85,B 0,C 180,E1 -13630.688,E2 -13630.688} C_VEL
LIN {X 0,Y 350.006,Z 295.854,A -85,B 0,C 180,E1 -13631.141,E2 -13631.141} C_VEL
LIN {X 0,Y 348.265,Z 293.421,A -85,B 0,C 180,E1 -13631.459,E2 -13631.459} C_VEL
LIN {X 0,Y 347.75,Z 291.477,A -85,B 0,C 180,E1 -13631.603,E2 -13631.603} C_VEL
LIN {X 0,Y 347.704,Z 291.477,A -85,B 0,C 180,E1 -13635.026,E2 -13635.026} C_VEL
LIN {X 0,Y 347.749,Z 291.471,A -85,B 0,C 180,E1 -13638.397,E2 -13638.397} C_VEL
LIN {X 0,Y 347.772,Z 291.47,A -85,B 0,C 180,E1 -13642.011,E2 -13642.011} C_VEL
LIN {X 0,Y 347.743,Z 291.48,A -85,B 0,C 180,E1 -13645.536,E2 -13645.536} C_VEL
LIN {X 0,Y 347.743,Z 291.47,A -85,B 0,C 180,E1 -13648.3,E2 -13648.3} C_VEL
LIN {X 0,Y 347.777,Z 291.467,A -85,B 0,C 180,E1 -13650.987,E2 -13650.987} C_VEL
LIN {X 0,Y 347.829,Z 291.459,A -85,B 0,C 180,E1 -13653.607,E2 -13653.607} C_VEL
LIN {X 0,Y 347.787,Z 291.472,A -85,B 0,C 180,E1 -13656.162,E2 -13656.162} C_VEL
LIN {X 0,Y 347.811,Z 291.47,A -85,B 0,C 180,E1 -13659.909,E2 -13659.909} C_VEL
LIN {X 0,Y 347.864,Z 291.456,A -85,B 0,C 180,E1 -13662.359,E2 -13662.359} C_VEL
LIN {X 0,Y 347.895,Z 291.458,A -85,B 0,C 180,E1 -13665.971,E2 -13665.971} C_VEL
LIN {X 0,Y 347.926,Z 291.436,A -85,B 0,C 180,E1 -13669.525,E2 -13669.525} C_VEL
LIN {X 0,Y 348.072,Z 291.425,A -85,B 0,C 180,E1 -13671.875,E2 -13671.875} C_VEL
LIN {X 0,Y 348.065,Z 291.44,A -85,B 0,C 180,E1 -13674.205,E2 -13674.205} C_VEL
LIN {X 0,Y 348.204,Z 291.397,A -85,B 0,C 180,E1 -13677.686,E2 -13677.686} C_VEL
LIN {X 0,Y 348.344,Z 291.404,A -85,B 0,C 180,E1 -13680,E2 -13680} C_VEL
LIN {X 0,Y 348.205,Z 291.411,A -85,B 0,C 180,E1 -13682.313,E2 -13682.313} C_VEL
LIN {X 0,Y 348.104,Z 291.437,A -85,B 0,C 180,E1 -13686.957,E2 -13686.957} C_VEL
LIN {X 0,Y 347.965,Z 291.437,A -85,B 0,C 180,E1 -13689.298,E2 -13689.298} C_VEL
LIN {X 0,Y 347.887,Z 291.459,A -85,B 0,C 180,E1 -13692.839,E2 -13692.839} C_VEL
LIN {X 0,Y 347.836,Z 291.468,A -85,B 0,C 180,E1 -13696.431,E2 -13696.431} C_VEL
LIN {X 0,Y 347.853,Z 291.465,A -85,B 0,C 180,E1 -13698.86,E2 -13698.86} C_VEL
LIN {X 0,Y 347.771,Z 291.479,A -85,B 0,C 180,E1 -13702.579,E2 -13702.579} C_VEL
LIN {X 0,Y 347.81,Z 291.474,A -85,B 0,C 180,E1 -13705.108,E2 -13705.108} C_VEL
LIN {X 0,Y 347.808,Z 291.473,A -85,B 0,C 180,E1 -13707.694,E2 -13707.694} C_VEL
LIN {X 0,Y 347.761,Z 291.479,A -85,B 0,C 180,E1 -13710.346,E2 -13710.346} C_VEL
LIN {X 0,Y 347.742,Z 291.489,A -85,B 0,C 180,E1 -13714.464,E2 -13714.464} C_VEL
LIN {X 0,Y 347.771,Z 291.483,A -85,B 0,C 180,E1 -13717.989,E2 -13717.989} C_VEL
LIN {X 0,Y 347.748,Z 291.486,A -85,B 0,C 180,E1 -13721.83,E2 -13721.83} C_VEL
LIN {X 0,Y 347.738,Z 291.485,A -85,B 0,C 180,E1 -13726.002,E2 -13726.002} C_VEL
LIN {X 0,Y 352.981,Z 305.284,A -85,B 0,C 180,E1 -13729.165,E2 -13729.165} C_VEL
LIN {X 0,Y 362.006,Z 321.27,A -85,B 0,C 180,E1 -13730.781,E2 -13730.781} C_VEL
LIN {X 0,Y 369.268,Z 334.845,A -85,B 0,C 180,E1 -13732.017,E2 -13732.017} C_VEL
LIN {X 0,Y 377.092,Z 351.273,A -85,B 0,C 180,E1 -13733.316,E2 -13733.316} C_VEL
LIN {X 0,Y 377.35,Z 354.415,A -85,B 0,C 180,E1 -13733.417,E2 -13733.417} C_VEL
LIN {X 0,Y 372.148,Z 512.536,A -85,B 0,C 180,E1 -13736.515,E2 -13736.515} C_VEL
LIN {X 0,Y 370.946,Z 528.492,A -85,B 0,C 180,E1 -13736.996,E2 -13736.996} C_VEL
LIN {X 0,Y 369.25,Z 545.227,A -85,B 0,C 180,E1 -13737.716,E2 -13737.716} C_VEL
LIN {X 0,Y 367.407,Z 560.403,A -85,B 0,C 180,E1 -13738.584,E2 -13738.584} C_VEL
LIN {X 0,Y 365.202,Z 575.371,A -85,B 0,C 180,E1 -13739.658,E2 -13739.658} C_VEL
LIN {X 0,Y 362.813,Z 589.598,A -85,B 0,C 180,E1 -13740.92,E2 -13740.92} C_VEL
LIN {X 0,Y 360.202,Z 603.452,A -85,B 0,C 180,E1 -13742.394,E2 -13742.394} C_VEL
LIN {X 0,Y 357.624,Z 616.59,A -85,B 0,C 180,E1 -13744.071,E2 -13744.071} C_VEL
LIN {X 0,Y 355.445,Z 627.83,A -85,B 0,C 180,E1 -13745.778,E2 -13745.778} C_VEL
LIN {X 0,Y 353.166,Z 639.04,A -85,B 0,C 180,E1 -13747.784,E2 -13747.784} C_VEL
LIN {X 0,Y 350.997,Z 649.91,A -85,B 0,C 180,E1 -13750.1,E2 -13750.1} C_VEL
LIN {X 0,Y 349.341,Z 659.054,A -85,B 0,C 180,E1 -13752.436,E2 -13752.436} C_VEL
LIN {X 0,Y 348.052,Z 666.721,A -85,B 0,C 180,E1 -13754.782,E2 -13754.782} C_VEL
LIN {X 0,Y 347.194,Z 672.986,A -85,B 0,C 180,E1 -13757.135,E2 -13757.135} C_VEL
LIN {X 0,Y 346.524,Z 678.12,A -85,B 0,C 180,E1 -13759.483,E2 -13759.483} C_VEL
LIN {X 0,Y 346.269,Z 682.119,A -85,B 0,C 180,E1 -13761.832,E2 -13761.832} C_VEL
LIN {X 0,Y 346.178,Z 685.08,A -85,B 0,C 180,E1 -13764.174,E2 -13764.174} C_VEL
LIN {X 0,Y 346.12,Z 687.029,A -85,B 0,C 180,E1 -13766.508,E2 -13766.508} C_VEL
LIN {X 0,Y 346.112,Z 687.995,A -85,B 0,C 180,E1 -13768.837,E2 -13768.837} C_VEL
LIN {X 0,Y 346.112,Z 687.993,A -85,B 0,C 180,E1 -13771.164,E2 -13771.164} C_VEL
LIN {X 0,Y 346.12,Z 687.02,A -85,B 0,C 180,E1 -13773.492,E2 -13773.492} C_VEL
LIN {X 0,Y 346.194,Z 685.01,A -85,B 0,C 180,E1 -13775.885,E2 -13775.885} C_VEL
LIN {X 0,Y 346.269,Z 682.103,A -85,B 0,C 180,E1 -13778.168,E2 -13778.168} C_VEL
LIN {X 0,Y 346.524,Z 678.103,A -85,B 0,C 180,E1 -13780.517,E2 -13780.517} C_VEL
LIN {X 0,Y 347.184,Z 672.959,A -85,B 0,C 180,E1 -13782.866,E2 -13782.866} C_VEL
LIN {X 0,Y 348.051,Z 666.684,A -85,B 0,C 180,E1 -13785.218,E2 -13785.218} C_VEL
LIN {X 0,Y 349.568,Z 657.993,A -85,B 0,C 180,E1 -13787.854,E2 -13787.854} C_VEL
LIN {X 0,Y 351.244,Z 648.614,A -85,B 0,C 180,E1 -13790.191,E2 -13790.191} C_VEL
LIN {X 0,Y 353.189,Z 638.974,A -85,B 0,C 180,E1 -13792.214,E2 -13792.214} C_VEL
LIN {X 0,Y 355.492,Z 627.747,A -85,B 0,C 180,E1 -13794.219,E2 -13794.219} C_VEL
LIN {X 0,Y 357.634,Z 616.496,A -85,B 0,C 180,E1 -13795.928,E2 -13795.928} C_VEL
LIN {X 0,Y 360.189,Z 603.337,A -85,B 0,C 180,E1 -13797.607,E2 -13797.607} C_VEL
LIN {X 0,Y 362.867,Z 588.732,A -85,B 0,C 180,E1 -13799.155,E2 -13799.155} C_VEL
LIN {X 0,Y 365.193,Z 575.185,A -85,B 0,C 180,E1 -13800.343,E2 -13800.343} C_VEL
LIN {X 0,Y 367.392,Z 560.19,A -85,B 0,C 180,E1 -13801.418,E2 -13801.418} C_VEL
LIN {X 0,Y 369.242,Z 544.957,A -85,B 0,C 180,E1 -13802.285,E2 -13802.285} C_VEL
LIN {X 0,Y 370.859,Z 529.028,A -85,B 0,C 180,E1 -13802.972,E2 -13802.972} C_VEL
LIN {X 0,Y 372.141,Z 513.379,A -85,B 0,C 180,E1 -13803.446,E2 -13803.446} C_VEL
LIN {X 0,Y 377.317,Z 353.608,A -85,B 0,C 180,E1 -13806.586,E2 -13806.586} C_VEL
LIN {X 0,Y 376.74,Z 350.598,A -85,B 0,C 180,E1 -13806.721,E2 -13806.721} C_VEL
LIN {X 0,Y 367.95,Z 332.267,A -85,B 0,C 180,E1 -13808.184,E2 -13808.184} C_VEL
LIN {X 0,Y 357.77,Z 313.591,A -85,B 0,C 180,E1 -13809.942,E2 -13809.942} C_VEL
LIN {X 0,Y 352.758,Z 304.867,A -85,B 0,C 180,E1 -13810.876,E2 -13810.876} C_VEL
LIN {X 0,Y 348.442,Z 293.754,A -85,B 0,C 180,E1 -13813.439,E2 -13813.439} C_VEL
LIN {X 0,Y 347.745,Z 291.477,A -85,B 0,C 180,E1 -13813.992,E2 -13813.992} C_VEL
LIN {X 0,Y 347.748,Z 291.472,A -85,B 0,C 180,E1 -13818.17,E2 -13818.17} C_VEL
LIN {X 0,Y 347.771,Z 291.471,A -85,B 0,C 180,E1 -13822.011,E2 -13822.011} C_VEL
LIN {X 0,Y 347.742,Z 291.476,A -85,B 0,C 180,E1 -13825.536,E2 -13825.536} C_VEL
LIN {X 0,Y 347.762,Z 291.473,A -85,B 0,C 180,E1 -13829.654,E2 -13829.654} C_VEL
LIN {X 0,Y 347.849,Z 291.464,A -85,B 0,C 180,E1 -13832.745,E2 -13832.745} C_VEL
LIN {X 0,Y 347.787,Z 291.473,A -85,B 0,C 180,E1 -13836.162,E2 -13836.162} C_VEL
LIN {X 0,Y 347.812,Z 291.444,A -85,B 0,C 180,E1 -13839.91,E2 -13839.91} C_VEL
LIN {X 0,Y 347.864,Z 291.462,A -85,B 0,C 180,E1 -13842.359,E2 -13842.359} C_VEL
LIN {X 0,Y 347.895,Z 291.433,A -85,B 0,C 180,E1 -13845.971,E2 -13845.971} C_VEL
LIN {X 0,Y 347.926,Z 291.459,A -85,B 0,C 180,E1 -13849.526,E2 -13849.526} C_VEL
LIN {X 0,Y 348.09,Z 291.407,A -85,B 0,C 180,E1 -13853.042,E2 -13853.042} C_VEL
LIN {X 0,Y 348.206,Z 291.421,A -85,B 0,C 180,E1 -13857.687,E2 -13857.687} C_VEL
LIN {X 0,Y 348.323,Z 291.381,A -85,B 0,C 180,E1 -13860,E2 -13860} C_VEL
LIN {X 0,Y 348.204,Z 291.405,A -85,B 0,C 180,E1 -13862.314,E2 -13862.314} C_VEL
LIN {X 0,Y 348.09,Z 291.412,A -85,B 0,C 180,E1 -13866.958,E2 -13866.958} C_VEL
LIN {X 0,Y 347.927,Z 291.45,A -85,B 0,C 180,E1 -13870.475,E2 -13870.475} C_VEL
LIN {X 0,Y 347.897,Z 291.44,A -85,B 0,C 180,E1 -13874.15,E2 -13874.15} C_VEL
LIN {X 0,Y 347.889,Z 291.462,A -85,B 0,C 180,E1 -13878.29,E2 -13878.29} C_VEL
LIN {X 0,Y 347.776,Z 291.448,A -85,B 0,C 180,E1 -13881.631,E2 -13881.631} C_VEL
LIN {X 0,Y 347.811,Z 291.474,A -85,B 0,C 180,E1 -13885.109,E2 -13885.109} C_VEL
LIN {X 0,Y 347.807,Z 291.447,A -85,B 0,C 180,E1 -13887.694,E2 -13887.694} C_VEL
LIN {X 0,Y 347.759,Z 291.478,A -85,B 0,C 180,E1 -13890.347,E2 -13890.347} C_VEL
LIN {X 0,Y 347.743,Z 291.476,A -85,B 0,C 180,E1 -13894.464,E2 -13894.464} C_VEL
LIN {X 0,Y 347.772,Z 291.456,A -85,B 0,C 180,E1 -13897.989,E2 -13897.989} C_VEL
LIN {X 0,Y 347.749,Z 291.464,A -85,B 0,C 180,E1 -13901.831,E2 -13901.831} C_VEL
LIN {X 0,Y 347.705,Z 291.477,A -85,B 0,C 180,E1 -13905.027,E2 -13905.027} C_VEL
LIN {X 0,Y 347.751,Z 291.48,A -85,B 0,C 180,E1 -13908.512,E2 -13908.512} C_VEL
LIN {X 0,Y 348.832,Z 294.475,A -85,B 0,C 180,E1 -13908.77,E2 -13908.77} C_VEL
LIN {X 0,Y 350.711,Z 296.799,A -85,B 0,C 180,E1 -13909.103,E2 -13909.103} C_VEL
LIN {X 0,Y 352.808,Z 300.03,A -85,B 0,C 180,E1 -13909.485,E2 -13909.485} C_VEL
LIN {X 0,Y 362.109,Z 314.494,A -85,B 0,C 180,E1 -13911.104,E2 -13911.104} C_VEL
LIN {X 0,Y 370.263,Z 329.259,A -85,B 0,C 180,E1 -13912.479,E2 -13912.479} C_VEL
LIN {X 0,Y 377.448,Z 343.746,A -85,B 0,C 180,E1 -13913.655,E2 -13913.655} C_VEL
LIN {X 0,Y 372.629,Z 493.674,A -85,B 0,C 180,E1 -13916.607,E2 -13916.607} C_VEL
LIN {X 0,Y 371.557,Z 509.815,A -85,B 0,C 180,E1 -13917.098,E2 -13917.098} C_VEL
LIN {X 0,Y 370.081,Z 525.974,A -85,B 0,C 180,E1 -13917.797,E2 -13917.797} C_VEL
LIN {X 0,Y 368.285,Z 541.295,A -85,B 0,C 180,E1 -13918.667,E2 -13918.667} C_VEL
LIN {X 0,Y 366.263,Z 555.741,A -85,B 0,C 180,E1 -13919.709,E2 -13919.709} C_VEL
LIN {X 0,Y 364.065,Z 570.107,A -85,B 0,C 180,E1 -13920.986,E2 -13920.986} C_VEL
LIN {X 0,Y 361.746,Z 583.153,A -85,B 0,C 180,E1 -13922.365,E2 -13922.365} C_VEL
LIN {X 0,Y 359.344,Z 595.375,A -85,B 0,C 180,E1 -13923.894,E2 -13923.894} C_VEL
LIN {X 0,Y 357.051,Z 606.749,A -85,B 0,C 180,E1 -13925.585,E2 -13925.585} C_VEL
LIN {X 0,Y 354.673,Z 618.153,A -85,B 0,C 180,E1 -13927.577,E2 -13927.577} C_VEL
LIN {X 0,Y 352.612,Z 628.277,A -85,B 0,C 180,E1 -13929.674,E2 -13929.674} C_VEL
LIN {X 0,Y 350.545,Z 638.379,A -85,B 0,C 180,E1 -13932.197,E2 -13932.197} C_VEL
LIN {X 0,Y 348.926,Z 646.911,A -85,B 0,C 180,E1 -13934.821,E2 -13934.821} C_VEL
LIN {X 0,Y 347.636,Z 654.474,A -85,B 0,C 180,E1 -13937.744,E2 -13937.744} C_VEL
LIN {X 0,Y 346.839,Z 660.212,A -85,B 0,C 180,E1 -13940.671,E2 -13940.671} C_VEL
LIN {X 0,Y 346.401,Z 664.534,A -85,B 0,C 180,E1 -13943.796,E2 -13943.796} C_VEL
LIN {X 0,Y 346.191,Z 666.814,A -85,B 0,C 180,E1 -13946.508,E2 -13946.508} C_VEL
LIN {X 0,Y 346.15,Z 667.779,A -85,B 0,C 180,E1 -13948.837,E2 -13948.837} C_VEL
LIN {X 0,Y 346.15,Z 667.793,A -85,B 0,C 180,E1 -13951.163,E2 -13951.163} C_VEL
LIN {X 0,Y 346.191,Z 666.884,A -85,B 0,C 180,E1 -13953.492,E2 -13953.492} C_VEL
LIN {X 0,Y 346.401,Z 664.646,A -85,B 0,C 180,E1 -13956.204,E2 -13956.204} C_VEL
LIN {X 0,Y 346.828,Z 660.389,A -85,B 0,C 180,E1 -13959.329,E2 -13959.329} C_VEL
LIN {X 0,Y 347.613,Z 654.702,A -85,B 0,C 180,E1 -13962.256,E2 -13962.256} C_VEL
LIN {X 0,Y 348.882,Z 647.216,A -85,B 0,C 180,E1 -13965.181,E2 -13965.181} C_VEL
LIN {X 0,Y 349.539,Z 643.62,A -85,B 0,C 180,E1 -13966.356,E2 -13966.356} C_VEL
LIN {X 0,Y 349.454,Z 640.886,A -85,B 0,C 180,E1 -13967.214,E2 -13967.214} C_VEL
LIN {X 0,Y 346.177,Z 632.68,A -85,B 0,C 180,E1 -13969.775,E2 -13969.775} C_VEL
LIN {X 0,Y 345.815,Z 629.513,A -85,B 0,C 180,E1 -13970.602,E2 -13970.602} C_VEL
LIN {X 0,Y 345.945,Z 628.373,A -85,B 0,C 180,E1 -13970.868,E2 -13970.868} C_VEL
LIN {X 0,Y 348.343,Z 617.388,A -85,B 0,C 180,E1 -13973.167,E2 -13973.167} C_VEL
LIN {X 0,Y 350.775,Z 606.055,A -85,B 0,C 180,E1 -13975.151,E2 -13975.151} C_VEL
LIN {X 0,Y 353.541,Z 593.108,A -85,B 0,C 180,E1 -13977.047,E2 -13977.047} C_VEL
LIN {X 0,Y 356.2,Z 579.244,A -85,B 0,C 180,E1 -13978.746,E2 -13978.746} C_VEL
LIN {X 0,Y 358.69,Z 565.939,A -85,B 0,C 180,E1 -13980.095,E2 -13980.095} C_VEL
LIN {X 0,Y 360.687,Z 552.886,A -85,B 0,C 180,E1 -13981.202,E2 -13981.202} C_VEL
LIN {X 0,Y 362.851,Z 537.463,A -85,B 0,C 180,E1 -13982.266,E2 -13982.266} C_VEL
LIN {X 0,Y 364.593,Z 521.861,A -85,B 0,C 180,E1 -13983.117,E2 -13983.117} C_VEL
LIN {X 0,Y 365.926,Z 506.951,A -85,B 0,C 180,E1 -13983.722,E2 -13983.722} C_VEL
LIN {X 0,Y 366.94,Z 490.449,A -85,B 0,C 180,E1 -13984.185,E2 -13984.185} C_VEL
LIN {X 0,Y 371.758,Z 346.174,A -85,B 0,C 180,E1 -13987.051,E2 -13987.051} C_VEL
LIN {X 0,Y 361.852,Z 326.606,A -85,B 0,C 180,E1 -13988.739,E2 -13988.739} C_VEL
LIN {X 0,Y 354.771,Z 314.507,A -85,B 0,C 180,E1 -13989.982,E2 -13989.982} C_VEL
LIN {X 0,Y 347.669,Z 303.786,A -85,B 0,C 180,E1 -13991.266,E2 -13991.266} C_VEL
LIN {X 0,Y 345.608,Z 300.665,A -85,B 0,C 180,E1 -13991.654,E2 -13991.654} C_VEL
LIN {X 0,Y 343.095,Z 296.825,A -85,B 0,C 180,E1 -13992.137,E2 -13992.137} C_VEL
LIN {X 0,Y 341.345,Z 294.62,A -85,B 0,C 180,E1 -13992.467,E2 -13992.467} C_VEL
LIN {X 0,Y 340.678,Z 292.352,A -85,B 0,C 180,E1 -13992.645,E2 -13992.645} C_VEL
LIN {X 0,Y 340.65,Z 292.356,A -85,B 0,C 180,E1 -13996.227,E2 -13996.227} C_VEL
LIN {X 0,Y 340.686,Z 292.351,A -85,B 0,C 180,E1 -13999.753,E2 -13999.753} C_VEL
LIN {X 0,Y 340.703,Z 292.344,A -85,B 0,C 180,E1 -14003.258,E2 -14003.258} C_VEL
LIN {X 0,Y 340.69,Z 292.353,A -85,B 0,C 180,E1 -14006.153,E2 -14006.153} C_VEL
LIN {X 0,Y 340.74,Z 292.353,A -85,B 0,C 180,E1 -14010.329,E2 -14010.329} C_VEL
LIN {X 0,Y 340.801,Z 292.327,A -85,B 0,C 180,E1 -14013.02,E2 -14013.02} C_VEL
LIN {X 0,Y 340.754,Z 292.349,A -85,B 0,C 180,E1 -14015.638,E2 -14015.638} C_VEL
LIN {X 0,Y 340.743,Z 292.342,A -85,B 0,C 180,E1 -14019.474,E2 -14019.474} C_VEL
LIN {X 0,Y 340.855,Z 292.334,A -85,B 0,C 180,E1 -14021.984,E2 -14021.984} C_VEL
LIN {X 0,Y 340.867,Z 292.327,A -85,B 0,C 180,E1 -14025.705,E2 -14025.705} C_VEL
LIN {X 0,Y 340.868,Z 292.317,A -85,B 0,C 180,E1 -14029.306,E2 -14029.306} C_VEL
LIN {X 0,Y 341.074,Z 292.307,A -85,B 0,C 180,E1 -14032.898,E2 -14032.898} C_VEL
LIN {X 0,Y 341.165,Z 292.273,A -85,B 0,C 180,E1 -14037.639,E2 -14037.639} C_VEL
LIN {X 0,Y 341.294,Z 292.283,A -85,B 0,C 180,E1 -14040,E2 -14040} C_VEL
LIN {X 0,Y 341.167,Z 292.286,A -85,B 0,C 180,E1 -14042.361,E2 -14042.361} C_VEL
LIN {X 0,Y 341.073,Z 292.314,A -85,B 0,C 180,E1 -14047.102,E2 -14047.102} C_VEL
LIN {X 0,Y 340.868,Z 292.311,A -85,B 0,C 180,E1 -14050.694,E2 -14050.694} C_VEL
LIN {X 0,Y 340.86,Z 292.339,A -85,B 0,C 180,E1 -14054.325,E2 -14054.325} C_VEL
LIN {X 0,Y 340.835,Z 292.337,A -85,B 0,C 180,E1 -14058.467,E2 -14058.467} C_VEL
LIN {X 0,Y 340.751,Z 292.35,A -85,B 0,C 180,E1 -14061.857,E2 -14061.857} C_VEL
LIN {X 0,Y 340.77,Z 292.353,A -85,B 0,C 180,E1 -14065.664,E2 -14065.664} C_VEL
LIN {X 0,Y 340.738,Z 292.356,A -85,B 0,C 180,E1 -14068.32,E2 -14068.32} C_VEL
LIN {X 0,Y 340.701,Z 292.362,A -85,B 0,C 180,E1 -14071.044,E2 -14071.044} C_VEL
LIN {X 0,Y 340.715,Z 292.357,A -85,B 0,C 180,E1 -14075.279,E2 -14075.279} C_VEL
LIN {X 0,Y 340.708,Z 292.365,A -85,B 0,C 180,E1 -14078.386,E2 -14078.386} C_VEL
LIN {X 0,Y 340.696,Z 292.365,A -85,B 0,C 180,E1 -14082.045,E2 -14082.045} C_VEL
LIN {X 0,Y 340.683,Z 292.504,A -85,B 0,C 180,E1 -14085.101,E2 -14085.101} C_VEL
LIN {X 0,Y 345.411,Z 304.861,A -85,B 0,C 180,E1 -14088.066,E2 -14088.066} C_VEL
LIN {X 0,Y 352.54,Z 316.912,A -85,B 0,C 180,E1 -14089.408,E2 -14089.408} C_VEL
LIN {X 0,Y 361.725,Z 333.699,A -85,B 0,C 180,E1 -14091.056,E2 -14091.056} C_VEL
LIN {X 0,Y 370.666,Z 352.148,A -85,B 0,C 180,E1 -14092.598,E2 -14092.598} C_VEL
LIN {X 0,Y 371.617,Z 354.226,A -85,B 0,C 180,E1 -14092.758,E2 -14092.758} C_VEL
LIN {X 0,Y 368.469,Z 445.563,A -85,B 0,C 180,E1 -14094.553,E2 -14094.553} C_VEL
LIN {X 0,Y 366.22,Z 513.005,A -85,B 0,C 180,E1 -14095.917,E2 -14095.917} C_VEL
LIN {X 0,Y 364.852,Z 530.129,A -85,B 0,C 180,E1 -14096.455,E2 -14096.455} C_VEL
LIN {X 0,Y 363.08,Z 546.33,A -85,B 0,C 180,E1 -14097.182,E2 -14097.182} C_VEL
LIN {X 0,Y 361.039,Z 562.191,A -85,B 0,C 180,E1 -14098.129,E2 -14098.129} C_VEL
LIN {X 0,Y 358.765,Z 576.829,A -85,B 0,C 180,E1 -14099.218,E2 -14099.218} C_VEL
LIN {X 0,Y 356.124,Z 591.865,A -85,B 0,C 180,E1 -14100.601,E2 -14100.601} C_VEL
LIN {X 0,Y 353.369,Z 605.603,A -85,B 0,C 180,E1 -14102.136,E2 -14102.136} C_VEL
LIN {X 0,Y 350.746,Z 618.345,A -85,B 0,C 180,E1 -14103.844,E2 -14103.844} C_VEL
LIN {X 0,Y 348.2,Z 630.992,A -85,B 0,C 180,E1 -14105.876,E2 -14105.876} C_VEL
LIN {X 0,Y 345.865,Z 641.774,A -85,B 0,C 180,E1 -14107.919,E2 -14107.919} C_VEL
LIN {X 0,Y 343.712,Z 652.205,A -85,B 0,C 180,E1 -14110.288,E2 -14110.288} C_VEL
LIN {X 0,Y 342.053,Z 660.88,A -85,B 0,C 180,E1 -14112.667,E2 -14112.667} C_VEL
LIN {X 0,Y 340.857,Z 668.164,A -85,B 0,C 180,E1 -14115.065,E2 -14115.065} C_VEL
LIN {X 0,Y 339.984,Z 674.211,A -85,B 0,C 180,E1 -14117.464,E2 -14117.464} C_VEL
LIN {X 0,Y 339.306,Z 680.074,A -85,B 0,C 180,E1 -14120.462,E2 -14120.462} C_VEL
LIN {X 0,Y 339.126,Z 683.508,A -85,B 0,C 180,E1 -14122.857,E2 -14122.857} C_VEL
LIN {X 0,Y 339.029,Z 686.004,A -85,B 0,C 180,E1 -14125.244,E2 -14125.244} C_VEL
LIN {X 0,Y 338.988,Z 687.412,A -85,B 0,C 180,E1 -14127.624,E2 -14127.624} C_VEL
LIN {X 0,Y 339.064,Z 687.943,A -85,B 0,C 180,E1 -14130,E2 -14130} C_VEL
LIN {X 0,Y 338.988,Z 687.406,A -85,B 0,C 180,E1 -14132.376,E2 -14132.376} C_VEL
LIN {X 0,Y 339.029,Z 685.992,A -85,B 0,C 180,E1 -14134.756,E2 -14134.756} C_VEL
LIN {X 0,Y 339.126,Z 683.492,A -85,B 0,C 180,E1 -14137.143,E2 -14137.143} C_VEL
LIN {X 0,Y 339.306,Z 680.055,A -85,B 0,C 180,E1 -14139.538,E2 -14139.538} C_VEL
LIN {X 0,Y 339.98,Z 674.185,A -85,B 0,C 180,E1 -14142.536,E2 -14142.536} C_VEL
LIN {X 0,Y 340.854,Z 668.129,A -85,B 0,C 180,E1 -14144.936,E2 -14144.936} C_VEL
LIN {X 0,Y 342.053,Z 660.834,A -85,B 0,C 180,E1 -14147.333,E2 -14147.333} C_VEL
LIN {X 0,Y 343.753,Z 652.065,A -85,B 0,C 180,E1 -14149.731,E2 -14149.731} C_VEL
LIN {X 0,Y 345.867,Z 641.71,A -85,B 0,C 180,E1 -14152.081,E2 -14152.081} C_VEL
LIN {X 0,Y 348.245,Z 630.913,A -85,B 0,C 180,E1 -14154.121,E2 -14154.121} C_VEL
LIN {X 0,Y 350.391,Z 620.21,A -85,B 0,C 180,E1 -14155.865,E2 -14155.865} C_VEL
LIN {X 0,Y 352.93,Z 607.816,A -85,B 0,C 180,E1 -14157.58,E2 -14157.58} C_VEL
LIN {X 0,Y 355.565,Z 594.353,A -85,B 0,C 180,E1 -14159.126,E2 -14159.126} C_VEL
LIN {X 0,Y 358.02,Z 580.96,A -85,B 0,C 180,E1 -14160.41,E2 -14160.41} C_VEL
LIN {X 0,Y 360.442,Z 565.949,A -85,B 0,C 180,E1 -14161.602,E2 -14161.602} C_VEL
LIN {X 0,Y 362.689,Z 549.938,A -85,B 0,C 180,E1 -14162.611,E2 -14162.611} C_VEL
LIN {X 0,Y 364.419,Z 533.924,A -85,B 0,C 180,E1 -14163.383,E2 -14163.383} C_VEL
LIN {X 0,Y 365.849,Z 518.203,A -85,B 0,C 180,E1 -14163.92,E2 -14163.92} C_VEL
LIN {X 0,Y 366.707,Z 500.56,A -85,B 0,C 180,E1 -14164.338,E2 -14164.338} C_VEL
LIN {X 0,Y 371.566,Z 354.942,A -85,B 0,C 180,E1 -14167.211,E2 -14167.211} C_VEL
LIN {X 0,Y 371.21,Z 353.363,A -85,B 0,C 180,E1 -14167.289,E2 -14167.289} C_VEL
LIN {X 0,Y 362.954,Z 336.174,A -85,B 0,C 180,E1 -14168.705,E2 -14168.705} C_VEL
LIN {X 0,Y 355.144,Z 321.626,A -85,B 0,C 180,E1 -14170.088,E2 -14170.088} C_VEL
LIN {X 0,Y 347.869,Z 308.914,A -85,B 0,C 180,E1 -14171.436,E2 -14171.436} C_VEL
LIN {X 0,Y 345.355,Z 304.715,A -85,B 0,C 180,E1 -14171.924,E2 -14171.924} C_VEL
LIN {X 0,Y 341.983,Z 296.01,A -85,B 0,C 180,E1 -14174.006,E2 -14174.006} C_VEL
LIN {X 0,Y 340.715,Z 292.353,A -85,B 0,C 180,E1 -14174.918,E2 -14174.918} C_VEL
LIN {X 0,Y 340.683,Z 292.353,A -85,B 0,C 180,E1 -14178.69,E2 -14178.69} C_VEL
LIN {X 0,Y 340.73,Z 292.349,A -85,B 0,C 180,E1 -14181.773,E2 -14181.773} C_VEL
LIN {X 0,Y 340.72,Z 292.351,A -85,B 0,C 180,E1 -14185.595,E2 -14185.595} C_VEL
LIN {X 0,Y 340.701,Z 292.358,A -85,B 0,C 180,E1 -14188.956,E2 -14188.956} C_VEL
LIN {X 0,Y 340.776,Z 292.345,A -85,B 0,C 180,E1 -14192.474,E2 -14192.474} C_VEL
LIN {X 0,Y 340.754,Z 292.348,A -85,B 0,C 180,E1 -14195.638,E2 -14195.638} C_VEL
LIN {X 0,Y 340.744,Z 292.326,A -85,B 0,C 180,E1 -14199.474,E2 -14199.474} C_VEL
LIN {X 0,Y 340.856,Z 292.333,A -85,B 0,C 180,E1 -14201.984,E2 -14201.984} C_VEL
LIN {X 0,Y 340.867,Z 292.31,A -85,B 0,C 180,E1 -14205.705,E2 -14205.705} C_VEL
LIN {X 0,Y 340.869,Z 292.336,A -85,B 0,C 180,E1 -14209.306,E2 -14209.306} C_VEL
LIN {X 0,Y 341.058,Z 292.283,A -85,B 0,C 180,E1 -14212.898,E2 -14212.898} C_VEL
LIN {X 0,Y 341.168,Z 292.298,A -85,B 0,C 180,E1 -14217.639,E2 -14217.639} C_VEL
LIN {X 0,Y 341.274,Z 292.258,A -85,B 0,C 180,E1 -14220,E2 -14220} C_VEL
LIN {X 0,Y 341.166,Z 292.282,A -85,B 0,C 180,E1 -14222.361,E2 -14222.361} C_VEL
LIN {X 0,Y 341.058,Z 292.285,A -85,B 0,C 180,E1 -14227.102,E2 -14227.102} C_VEL
LIN {X 0,Y 340.869,Z 292.331,A -85,B 0,C 180,E1 -14230.694,E2 -14230.694} C_VEL
LIN {X 0,Y 340.862,Z 292.313,A -85,B 0,C 180,E1 -14234.325,E2 -14234.325} C_VEL
LIN {X 0,Y 340.835,Z 292.341,A -85,B 0,C 180,E1 -14238.467,E2 -14238.467} C_VEL
LIN {X 0,Y 340.722,Z 292.325,A -85,B 0,C 180,E1 -14241.844,E2 -14241.844} C_VEL
LIN {X 0,Y 340.771,Z 292.347,A -85,B 0,C 180,E1 -14245.665,E2 -14245.665} C_VEL
LIN {X 0,Y 340.727,Z 292.33,A -85,B 0,C 180,E1 -14248.321,E2 -14248.321} C_VEL
LIN {X 0,Y 340.701,Z 292.357,A -85,B 0,C 180,E1 -14251.044,E2 -14251.044} C_VEL
LIN {X 0,Y 340.717,Z 292.354,A -85,B 0,C 180,E1 -14255.279,E2 -14255.279} C_VEL
LIN {X 0,Y 340.708,Z 292.336,A -85,B 0,C 180,E1 -14258.386,E2 -14258.386} C_VEL
LIN {X 0,Y 340.698,Z 292.341,A -85,B 0,C 180,E1 -14262.046,E2 -14262.046} C_VEL
LIN {X 0,Y 340.651,Z 292.351,A -85,B 0,C 180,E1 -14266.227,E2 -14266.227} C_VEL
LIN {X 0,Y 340.689,Z 292.362,A -85,B 0,C 180,E1 -14267.473,E2 -14267.473} C_VEL
LIN {X 0,Y 341.654,Z 295.164,A -85,B 0,C 180,E1 -14267.717,E2 -14267.717} C_VEL
LIN {X 0,Y 343.675,Z 297.582,A -85,B 0,C 180,E1 -14268.092,E2 -14268.092} C_VEL
LIN {X 0,Y 345.885,Z 301.018,A -85,B 0,C 180,E1 -14268.516,E2 -14268.516} C_VEL
LIN {X 0,Y 354.939,Z 314.835,A -85,B 0,C 180,E1 -14270.165,E2 -14270.165} C_VEL
LIN {X 0,Y 361.346,Z 325.828,A -85,B 0,C 180,E1 -14271.29,E2 -14271.29} C_VEL
LIN {X 0,Y 369.835,Z 342.248,A -85,B 0,C 180,E1 -14272.739,E2 -14272.739} C_VEL
LIN {X 0,Y 371.742,Z 346.199,A -85,B 0,C 180,E1 -14273.058,E2 -14273.058} C_VEL
LIN {X 0,Y 366.716,Z 494.109,A -85,B 0,C 180,E1 -14276.001,E2 -14276.001} C_VEL
LIN {X 0,Y 365.631,Z 510.035,A -85,B 0,C 180,E1 -14276.495,E2 -14276.495} C_VEL
LIN {X 0,Y 364.089,Z 526.191,A -85,B 0,C 180,E1 -14277.202,E2 -14277.202} C_VEL
LIN {X 0,Y 362.246,Z 541.509,A -85,B 0,C 180,E1 -14278.084,E2 -14278.084} C_VEL
LIN {X 0,Y 360.074,Z 556.491,A -85,B 0,C 180,E1 -14279.182,E2 -14279.182} C_VEL
LIN {X 0,Y 357.834,Z 570.32,A -85,B 0,C 180,E1 -14280.432,E2 -14280.432} C_VEL
LIN {X 0,Y 355.435,Z 583.366,A -85,B 0,C 180,E1 -14281.831,E2 -14281.831} C_VEL
LIN {X 0,Y 352.723,Z 596.732,A -85,B 0,C 180,E1 -14283.541,E2 -14283.541} C_VEL
LIN {X 0,Y 350.182,Z 608.731,A -85,B 0,C 180,E1 -14285.39,E2 -14285.39} C_VEL
LIN {X 0,Y 347.719,Z 619.839,A -85,B 0,C 180,E1 -14287.417,E2 -14287.417} C_VEL
LIN {X 0,Y 345.445,Z 630.578,A -85,B 0,C 180,E1 -14289.766,E2 -14289.766} C_VEL
LIN {X 0,Y 343.51,Z 639.594,A -85,B 0,C 180,E1 -14292.128,E2 -14292.128} C_VEL
LIN {X 0,Y 342.013,Z 647.122,A -85,B 0,C 180,E1 -14294.506,E2 -14294.506} C_VEL
LIN {X 0,Y 340.663,Z 654.683,A -85,B 0,C 180,E1 -14297.49,E2 -14297.49} C_VEL
LIN {X 0,Y 339.811,Z 660.421,A -85,B 0,C 180,E1 -14300.476,E2 -14300.476} C_VEL
LIN {X 0,Y 339.434,Z 663.78,A -85,B 0,C 180,E1 -14302.864,E2 -14302.864} C_VEL
LIN {X 0,Y 339.199,Z 666.221,A -85,B 0,C 180,E1 -14305.246,E2 -14305.246} C_VEL
LIN {X 0,Y 339.058,Z 667.608,A -85,B 0,C 180,E1 -14307.624,E2 -14307.624} C_VEL
LIN {X 0,Y 339.069,Z 668.142,A -85,B 0,C 180,E1 -14310,E2 -14310} C_VEL
LIN {X 0,Y 339.057,Z 667.65,A -85,B 0,C 180,E1 -14312.376,E2 -14312.376} C_VEL
LIN {X 0,Y 339.198,Z 666.303,A -85,B 0,C 180,E1 -14314.754,E2 -14314.754} C_VEL
LIN {X 0,Y 339.431,Z 663.904,A -85,B 0,C 180,E1 -14317.136,E2 -14317.136} C_VEL
LIN {X 0,Y 339.801,Z 660.596,A -85,B 0,C 180,E1 -14319.524,E2 -14319.524} C_VEL
LIN {X 0,Y 340.641,Z 654.909,A -85,B 0,C 180,E1 -14322.511,E2 -14322.511} C_VEL
LIN {X 0,Y 341.984,Z 647.423,A -85,B 0,C 180,E1 -14325.495,E2 -14325.495} C_VEL
LIN {X 0,Y 343.679,Z 638.936,A -85,B 0,C 180,E1 -14328.171,E2 -14328.171} C_VEL
LIN {X 0,Y 345.726,Z 629.498,A -85,B 0,C 180,E1 -14330.597,E2 -14330.597} C_VEL
LIN {X 0,Y 345.945,Z 628.373,A -85,B 0,C 180,E1 -14330.868,E2 -14330.868} C_VEL
LIN {X 0,Y 345.979,Z 624.985,A -85,B 0,C 180,E1 -14331.669,E2 -14331.669} C_VEL
LIN {X 0,Y 343.244,Z 613.636,A -85,B 0,C 180,E1 -14334.335,E2 -14334.335} C_VEL
LIN {X 0,Y 343.541,Z 609.756,A -85,B 0,C 180,E1 -14335.076,E2 -14335.076} C_VEL
LIN {X 0,Y 346.071,Z 598.459,A -85,B 0,C 180,E1 -14336.862,E2 -14336.862} C_VEL
LIN {X 0,Y 348.787,Z 585.517,A -85,B 0,C 180,E1 -14338.591,E2 -14338.591} C_VEL
LIN {X 0,Y 351.552,Z 571.624,A -85,B 0,C 180,E1 -14340.133,E2 -14340.133} C_VEL
LIN {X 0,Y 353.833,Z 557.841,A -85,B 0,C 180,E1 -14341.425,E2 -14341.425} C_VEL
LIN {X 0,Y 356.398,Z 541.026,A -85,B 0,C 180,E1 -14342.671,E2 -14342.671} C_VEL
LIN {X 0,Y 358.318,Z 525.503,A -85,B 0,C 180,E1 -14343.563,E2 -14343.563} C_VEL
LIN {X 0,Y 359.802,Z 509.888,A -85,B 0,C 180,E1 -14344.249,E2 -14344.249} C_VEL
LIN {X 0,Y 360.933,Z 493.702,A -85,B 0,C 180,E1 -14344.748,E2 -14344.748} C_VEL
LIN {X 0,Y 366.038,Z 348.507,A -85,B 0,C 180,E1 -14347.677,E2 -14347.677} C_VEL
LIN {X 0,Y 357.234,Z 331.085,A -85,B 0,C 180,E1 -14349.226,E2 -14349.226} C_VEL
LIN {X 0,Y 350.275,Z 319.071,A -85,B 0,C 180,E1 -14350.485,E2 -14350.485} C_VEL
LIN {X 0,Y 341.474,Z 305.712,A -85,B 0,C 180,E1 -14352.137,E2 -14352.137} C_VEL
LIN {X 0,Y 338.527,Z 301.502,A -85,B 0,C 180,E1 -14352.712,E2 -14352.712} C_VEL
LIN {X 0,Y 336.214,Z 297.89,A -85,B 0,C 180,E1 -14353.183,E2 -14353.183} C_VEL
LIN {X 0,Y 334.321,Z 295.558,A -85,B 0,C 180,E1 -14353.558,E2 -14353.558} C_VEL
LIN {X 0,Y 333.622,Z 293.24,A -85,B 0,C 180,E1 -14353.763,E2 -14353.763} C_VEL
LIN {X 0,Y 333.64,Z 293.237,A -85,B 0,C 180,E1 -14357.618,E2 -14357.618} C_VEL
LIN {X 0,Y 333.651,Z 293.237,A -85,B 0,C 180,E1 -14361.202,E2 -14361.202} C_VEL
LIN {X 0,Y 333.674,Z 293.223,A -85,B 0,C 180,E1 -14363.861,E2 -14363.861} C_VEL
LIN {X 0,Y 333.641,Z 293.22,A -85,B 0,C 180,E1 -14367.413,E2 -14367.413} C_VEL
LIN {X 0,Y 333.688,Z 293.221,A -85,B 0,C 180,E1 -14371.026,E2 -14371.026} C_VEL
LIN {X 0,Y 333.733,Z 293.216,A -85,B 0,C 180,E1 -14373.753,E2 -14373.753} C_VEL
LIN {X 0,Y 333.718,Z 293.203,A -85,B 0,C 180,E1 -14377.914,E2 -14377.914} C_VEL
LIN {X 0,Y 333.792,Z 293.216,A -85,B 0,C 180,E1 -14381.589,E2 -14381.589} C_VEL
LIN {X 0,Y 333.806,Z 293.203,A -85,B 0,C 180,E1 -14385.576,E2 -14385.576} C_VEL
LIN {X 0,Y 333.831,Z 293.196,A -85,B 0,C 180,E1 -14389.078,E2 -14389.078} C_VEL
LIN {X 0,Y 334.023,Z 293.184,A -85,B 0,C 180,E1 -14392.747,E2 -14392.747} C_VEL
LIN {X 0,Y 333.808,Z 293.207,A -85,B 0,C 180,E1 -14395.169,E2 -14395.169} C_VEL
LIN {X 0,Y 334.103,Z 293.152,A -85,B 0,C 180,E1 -14397.589,E2 -14397.589} C_VEL
LIN {X 0,Y 334.245,Z 293.161,A -85,B 0,C 180,E1 -14400,E2 -14400} C_VEL
LIN {X 0,Y 334.104,Z 293.164,A -85,B 0,C 180,E1 -14402.411,E2 -14402.411} C_VEL
LIN {X 0,Y 334.023,Z 293.191,A -85,B 0,C 180,E1 -14407.252,E2 -14407.252} C_VEL
LIN {X 0,Y 333.831,Z 293.187,A -85,B 0,C 180,E1 -14410.922,E2 -14410.922} C_VEL
LIN {X 0,Y 333.806,Z 293.215,A -85,B 0,C 180,E1 -14414.634,E2 -14414.634} C_VEL
LIN {X 0,Y 333.794,Z 293.215,A -85,B 0,C 180,E1 -14418.655,E2 -14418.655} C_VEL
LIN {X 0,Y 333.69,Z 293.231,A -85,B 0,C 180,E1 -14422.278,E2 -14422.278} C_VEL
LIN {X 0,Y 333.733,Z 293.231,A -85,B 0,C 180,E1 -14426.246,E2 -14426.246} C_VEL
LIN {X 0,Y 333.708,Z 293.235,A -85,B 0,C 180,E1 -14428.972,E2 -14428.972} C_VEL
LIN {X 0,Y 333.64,Z 293.24,A -85,B 0,C 180,E1 -14432.587,E2 -14432.587} C_VEL
LIN {X 0,Y 333.674,Z 293.235,A -85,B 0,C 180,E1 -14436.139,E2 -14436.139} C_VEL
LIN {X 0,Y 333.644,Z 293.245,A -85,B 0,C 180,E1 -14439.192,E2 -14439.192} C_VEL
LIN {X 0,Y 333.63,Z 293.245,A -85,B 0,C 180,E1 -14442.5,E2 -14442.5} C_VEL
LIN {X 0,Y 333.606,Z 293.349,A -85,B 0,C 180,E1 -14444.097,E2 -14444.097} C_VEL
LIN {X 0,Y 338.107,Z 304.826,A -85,B 0,C 180,E1 -14446.95,E2 -14446.95} C_VEL
LIN {X 0,Y 345.126,Z 316.402,A -85,B 0,C 180,E1 -14448.338,E2 -14448.338} C_VEL
LIN {X 0,Y 352.786,Z 330.086,A -85,B 0,C 180,E1 -14449.786,E2 -14449.786} C_VEL
LIN {X 0,Y 360.218,Z 344.384,A -85,B 0,C 180,E1 -14451.131,E2 -14451.131} C_VEL
LIN {X 0,Y 365.89,Z 356.486,A -85,B 0,C 180,E1 -14452.133,E2 -14452.133} C_VEL
LIN {X 0,Y 362.577,Z 448.958,A -85,B 0,C 180,E1 -14453.973,E2 -14453.973} C_VEL
LIN {X 0,Y 360.331,Z 513.419,A -85,B 0,C 180,E1 -14455.3,E2 -14455.3} C_VEL
LIN {X 0,Y 358.866,Z 530.849,A -85,B 0,C 180,E1 -14455.861,E2 -14455.861} C_VEL
LIN {X 0,Y 357.129,Z 546.13,A -85,B 0,C 180,E1 -14456.564,E2 -14456.564} C_VEL
LIN {X 0,Y 355.002,Z 561.989,A -85,B 0,C 180,E1 -14457.521,E2 -14457.521} C_VEL
LIN {X 0,Y 352.64,Z 576.625,A -85,B 0,C 180,E1 -14458.624,E2 -14458.624} C_VEL
LIN {X 0,Y 349.904,Z 591.66,A -85,B 0,C 180,E1 -14460.025,E2 -14460.025} C_VEL
LIN {X 0,Y 347.046,Z 605.397,A -85,B 0,C 180,E1 -14461.583,E2 -14461.583} C_VEL
LIN {X 0,Y 344.326,Z 618.138,A -85,B 0,C 180,E1 -14463.318,E2 -14463.318} C_VEL
LIN {X 0,Y 341.627,Z 630.806,A -85,B 0,C 180,E1 -14465.385,E2 -14465.385} C_VEL
LIN {X 0,Y 339.206,Z 641.565,A -85,B 0,C 180,E1 -14467.462,E2 -14467.462} C_VEL
LIN {X 0,Y 337.006,Z 651.651,A -85,B 0,C 180,E1 -14469.791,E2 -14469.791} C_VEL
LIN {X 0,Y 335.206,Z 660.671,A -85,B 0,C 180,E1 -14472.302,E2 -14472.302} C_VEL
LIN {X 0,Y 333.901,Z 667.954,A -85,B 0,C 180,E1 -14474.746,E2 -14474.746} C_VEL
LIN {X 0,Y 332.973,Z 674.003,A -85,B 0,C 180,E1 -14477.196,E2 -14477.196} C_VEL
LIN {X 0,Y 332.251,Z 679.866,A -85,B 0,C 180,E1 -14480.258,E2 -14480.258} C_VEL
LIN {X 0,Y 332.028,Z 683.299,A -85,B 0,C 180,E1 -14482.704,E2 -14482.704} C_VEL
LIN {X 0,Y 331.938,Z 685.796,A -85,B 0,C 180,E1 -14485.142,E2 -14485.142} C_VEL
LIN {X 0,Y 331.905,Z 687.205,A -85,B 0,C 180,E1 -14487.573,E2 -14487.573} C_VEL
LIN {X 0,Y 331.967,Z 687.736,A -85,B 0,C 180,E1 -14490,E2 -14490} C_VEL
LIN {X 0,Y 331.905,Z 687.199,A -85,B 0,C 180,E1 -14492.427,E2 -14492.427} C_VEL
LIN {X 0,Y 331.938,Z 685.784,A -85,B 0,C 180,E1 -14494.858,E2 -14494.858} C_VEL
LIN {X 0,Y 332.028,Z 683.283,A -85,B 0,C 180,E1 -14497.296,E2 -14497.296} C_VEL
LIN {X 0,Y 332.252,Z 679.845,A -85,B 0,C 180,E1 -14499.743,E2 -14499.743} C_VEL
LIN {X 0,Y 332.966,Z 673.974,A -85,B 0,C 180,E1 -14502.805,E2 -14502.805} C_VEL
LIN {X 0,Y 333.9,Z 667.917,A -85,B 0,C 180,E1 -14505.254,E2 -14505.254} C_VEL
LIN {X 0,Y 335.209,Z 660.623,A -85,B 0,C 180,E1 -14507.698,E2 -14507.698} C_VEL
LIN {X 0,Y 337.031,Z 651.54,A -85,B 0,C 180,E1 -14510.221,E2 -14510.221} C_VEL
LIN {X 0,Y 339.222,Z 641.498,A -85,B 0,C 180,E1 -14512.537,E2 -14512.537} C_VEL
LIN {X 0,Y 341.678,Z 630.755,A -85,B 0,C 180,E1 -14514.604,E2 -14514.604} C_VEL
LIN {X 0,Y 343.909,Z 619.997,A -85,B 0,C 180,E1 -14516.389,E2 -14516.389} C_VEL
LIN {X 0,Y 346.59,Z 607.604,A -85,B 0,C 180,E1 -14518.128,E2 -14518.128} C_VEL
LIN {X 0,Y 349.334,Z 594.141,A -85,B 0,C 180,E1 -14519.697,E2 -14519.697} C_VEL
LIN {X 0,Y 352.095,Z 579.507,A -85,B 0,C 180,E1 -14521.108,E2 -14521.108} C_VEL
LIN {X 0,Y 354.398,Z 565.736,A -85,B 0,C 180,E1 -14522.205,E2 -14522.205} C_VEL
LIN {X 0,Y 356.696,Z 549.722,A -85,B 0,C 180,E1 -14523.229,E2 -14523.229} C_VEL
LIN {X 0,Y 358.418,Z 534.471,A -85,B 0,C 180,E1 -14523.975,E2 -14523.975} C_VEL
LIN {X 0,Y 359.967,Z 518.118,A -85,B 0,C 180,E1 -14524.547,E2 -14524.547} C_VEL
LIN {X 0,Y 360.843,Z 500.647,A -85,B 0,C 180,E1 -14524.969,E2 -14524.969} C_VEL
LIN {X 0,Y 365.836,Z 356.443,A -85,B 0,C 180,E1 -14527.853,E2 -14527.853} C_VEL
LIN {X 0,Y 357.482,Z 339.037,A -85,B 0,C 180,E1 -14529.332,E2 -14529.332} C_VEL
LIN {X 0,Y 348.183,Z 321.737,A -85,B 0,C 180,E1 -14531.048,E2 -14531.048} C_VEL
LIN {X 0,Y 343.024,Z 312.942,A -85,B 0,C 180,E1 -14532.038,E2 -14532.038} C_VEL
LIN {X 0,Y 337.903,Z 304.432,A -85,B 0,C 180,E1 -14533.067,E2 -14533.067} C_VEL
LIN {X 0,Y 333.635,Z 293.232,A -85,B 0,C 180,E1 -14535.902,E2 -14535.902} C_VEL
LIN {X 0,Y 333.645,Z 293.235,A -85,B 0,C 180,E1 -14539.315,E2 -14539.315} C_VEL
LIN {X 0,Y 333.663,Z 293.228,A -85,B 0,C 180,E1 -14543.168,E2 -14543.168} C_VEL
LIN {X 0,Y 333.672,Z 293.227,A -85,B 0,C 180,E1 -14545.341,E2 -14545.341} C_VEL
LIN {X 0,Y 333.7,Z 293.224,A -85,B 0,C 180,E1 -14549.71,E2 -14549.71} C_VEL
LIN {X 0,Y 333.741,Z 293.221,A -85,B 0,C 180,E1 -14552.401,E2 -14552.401} C_VEL
LIN {X 0,Y 333.725,Z 293.224,A -85,B 0,C 180,E1 -14555.091,E2 -14555.091} C_VEL
LIN {X 0,Y 333.678,Z 293.209,A -85,B 0,C 180,E1 -14559.019,E2 -14559.019} C_VEL
LIN {X 0,Y 333.792,Z 293.204,A -85,B 0,C 180,E1 -14561.59,E2 -14561.59} C_VEL
LIN {X 0,Y 333.806,Z 293.19,A -85,B 0,C 180,E1 -14565.577,E2 -14565.577} C_VEL
LIN {X 0,Y 333.832,Z 293.209,A -85,B 0,C 180,E1 -14569.078,E2 -14569.078} C_VEL
LIN {X 0,Y 334.005,Z 293.162,A -85,B 0,C 180,E1 -14572.747,E2 -14572.747} C_VEL
LIN {X 0,Y 333.808,Z 293.197,A -85,B 0,C 180,E1 -14575.169,E2 -14575.169} C_VEL
LIN {X 0,Y 334.105,Z 293.178,A -85,B 0,C 180,E1 -14577.589,E2 -14577.589} C_VEL
LIN {X 0,Y 334.225,Z 293.134,A -85,B 0,C 180,E1 -14580,E2 -14580} C_VEL
LIN {X 0,Y 334.104,Z 293.161,A -85,B 0,C 180,E1 -14582.411,E2 -14582.411} C_VEL
LIN {X 0,Y 333.991,Z 293.172,A -85,B 0,C 180,E1 -14586.598,E2 -14586.598} C_VEL
LIN {X 0,Y 333.849,Z 293.19,A -85,B 0,C 180,E1 -14589.696,E2 -14589.696} C_VEL
LIN {X 0,Y 333.795,Z 293.206,A -85,B 0,C 180,E1 -14593.392,E2 -14593.392} C_VEL
LIN {X 0,Y 333.745,Z 293.212,A -85,B 0,C 180,E1 -14597.146,E2 -14597.146} C_VEL
LIN {X 0,Y 333.731,Z 293.221,A -85,B 0,C 180,E1 -14599.691,E2 -14599.691} C_VEL
LIN {X 0,Y 333.673,Z 293.221,A -85,B 0,C 180,E1 -14603.59,E2 -14603.59} C_VEL
LIN {X 0,Y 333.734,Z 293.216,A -85,B 0,C 180,E1 -14606.247,E2 -14606.247} C_VEL
LIN {X 0,Y 333.708,Z 293.21,A -85,B 0,C 180,E1 -14608.972,E2 -14608.972} C_VEL
LIN {X 0,Y 333.642,Z 293.233,A -85,B 0,C 180,E1 -14612.587,E2 -14612.587} C_VEL
LIN {X 0,Y 333.675,Z 293.232,A -85,B 0,C 180,E1 -14616.139,E2 -14616.139} C_VEL
LIN {X 0,Y 333.646,Z 293.222,A -85,B 0,C 180,E1 -14619.193,E2 -14619.193} C_VEL
LIN {X 0,Y 333.631,Z 293.221,A -85,B 0,C 180,E1 -14622.5,E2 -14622.5} C_VEL
LIN {X 0,Y 333.62,Z 293.227,A -85,B 0,C 180,E1 -14626.363,E2 -14626.363} C_VEL
LIN {X 0,Y 334.655,Z 296.152,A -85,B 0,C 180,E1 -14626.638,E2 -14626.638} C_VEL
LIN {X 0,Y 336.735,Z 298.577,A -85,B 0,C 180,E1 -14627.043,E2 -14627.043} C_VEL
LIN {X 0,Y 338.883,Z 301.908,A -85,B 0,C 180,E1 -14627.477,E2 -14627.477} C_VEL
LIN {X 0,Y 348.159,Z 315.784,A -85,B 0,C 180,E1 -14629.245,E2 -14629.245} C_VEL
LIN {X 0,Y 354.395,Z 326.059,A -85,B 0,C 180,E1 -14630.382,E2 -14630.382} C_VEL
LIN {X 0,Y 361.323,Z 339.053,A -85,B 0,C 180,E1 -14631.617,E2 -14631.617} C_VEL
LIN {X 0,Y 366.007,Z 348.544,A -85,B 0,C 180,E1 -14632.432,E2 -14632.432} C_VEL
LIN {X 0,Y 360.894,Z 493.732,A -85,B 0,C 180,E1 -14635.358,E2 -14635.358} C_VEL
LIN {X 0,Y 359.724,Z 510.255,A -85,B 0,C 180,E1 -14635.87,E2 -14635.87} C_VEL
LIN {X 0,Y 358.159,Z 526.406,A -85,B 0,C 180,E1 -14636.588,E2 -14636.588} C_VEL
LIN {X 0,Y 356.255,Z 541.722,A -85,B 0,C 180,E1 -14637.482,E2 -14637.482} C_VEL
LIN {X 0,Y 353.87,Z 557.422,A -85,B 0,C 180,E1 -14638.649,E2 -14638.649} C_VEL
LIN {X 0,Y 351.405,Z 571.953,A -85,B 0,C 180,E1 -14640.001,E2 -14640.001} C_VEL
LIN {X 0,Y 348.918,Z 584.745,A -85,B 0,C 180,E1 -14641.421,E2 -14641.421} C_VEL
LIN {X 0,Y 346.143,Z 597.816,A -85,B 0,C 180,E1 -14643.144,E2 -14643.144} C_VEL
LIN {X 0,Y 343.335,Z 610.679,A -85,B 0,C 180,E1 -14645.189,E2 -14645.189} C_VEL
LIN {X 0,Y 340.787,Z 621.525,A -85,B 0,C 180,E1 -14647.252,E2 -14647.252} C_VEL
LIN {X 0,Y 338.738,Z 630.789,A -85,B 0,C 180,E1 -14649.347,E2 -14649.347} C_VEL
LIN {X 0,Y 336.709,Z 639.804,A -85,B 0,C 180,E1 -14651.755,E2 -14651.755} C_VEL
LIN {X 0,Y 335.119,Z 647.333,A -85,B 0,C 180,E1 -14654.179,E2 -14654.179} C_VEL
LIN {X 0,Y 333.701,Z 654.893,A -85,B 0,C 180,E1 -14657.224,E2 -14657.224} C_VEL
LIN {X 0,Y 332.764,Z 660.631,A -85,B 0,C 180,E1 -14660.273,E2 -14660.273} C_VEL
LIN {X 0,Y 332.362,Z 663.989,A -85,B 0,C 180,E1 -14662.711,E2 -14662.711} C_VEL
LIN {X 0,Y 332.123,Z 666.429,A -85,B 0,C 180,E1 -14665.144,E2 -14665.144} C_VEL
LIN {X 0,Y 331.972,Z 667.815,A -85,B 0,C 180,E1 -14667.573,E2 -14667.573} C_VEL
LIN {X 0,Y 331.972,Z 668.349,A -85,B 0,C 180,E1 -14670,E2 -14670} C_VEL
LIN {X 0,Y 331.972,Z 667.857,A -85,B 0,C 180,E1 -14672.427,E2 -14672.427} C_VEL
LIN {X 0,Y 332.123,Z 666.51,A -85,B 0,C 180,E1 -14674.855,E2 -14674.855} C_VEL
LIN {X 0,Y 332.359,Z 664.111,A -85,B 0,C 180,E1 -14677.289,E2 -14677.289} C_VEL
LIN {X 0,Y 332.755,Z 660.804,A -85,B 0,C 180,E1 -14679.728,E2 -14679.728} C_VEL
LIN {X 0,Y 333.68,Z 655.117,A -85,B 0,C 180,E1 -14682.777,E2 -14682.777} C_VEL
LIN {X 0,Y 335.096,Z 647.63,A -85,B 0,C 180,E1 -14685.822,E2 -14685.822} C_VEL
LIN {X 0,Y 336.858,Z 639.144,A -85,B 0,C 180,E1 -14688.552,E2 -14688.552} C_VEL
LIN {X 0,Y 338.676,Z 631.198,A -85,B 0,C 180,E1 -14690.657,E2 -14690.657} C_VEL
LIN {X 0,Y 340.746,Z 622.016,A -85,B 0,C 180,E1 -14692.751,E2 -14692.751} C_VEL
LIN {X 0,Y 343.208,Z 611.22,A -85,B 0,C 180,E1 -14694.821,E2 -14694.821} C_VEL
LIN {X 0,Y 343.541,Z 609.756,A -85,B 0,C 180,E1 -14695.076,E2 -14695.076} C_VEL
LIN {X 0,Y 343.873,Z 605.77,A -85,B 0,C 180,E1 -14695.801,E2 -14695.801} C_VEL
LIN {X 0,Y 342.82,Z 599.293,A -85,B 0,C 180,E1 -14697.042,E2 -14697.042} C_VEL
LIN {X 0,Y 341.771,Z 592.491,A -85,B 0,C 180,E1 -14698.236,E2 -14698.236} C_VEL
LIN {X 0,Y 342.089,Z 587.998,A -85,B 0,C 180,E1 -14698.876,E2 -14698.876} C_VEL
LIN {X 0,Y 344.398,Z 577.077,A -85,B 0,C 180,E1 -14700.166,E2 -14700.166} C_VEL
LIN {X 0,Y 347.016,Z 562.459,A -85,B 0,C 180,E1 -14701.639,E2 -14701.639} C_VEL
LIN {X 0,Y 349.55,Z 547.185,A -85,B 0,C 180,E1 -14702.878,E2 -14702.878} C_VEL
LIN {X 0,Y 351.719,Z 532.183,A -85,B 0,C 180,E1 -14703.848,E2 -14703.848} C_VEL
LIN {X 0,Y 353.466,Z 515.409,A -85,B 0,C 180,E1 -14704.691,E2 -14704.691} C_VEL
LIN {X 0,Y 354.807,Z 499.579,A -85,B 0,C 180,E1 -14705.242,E2 -14705.242} C_VEL
LIN {X 0,Y 355.806,Z 477.298,A -85,B 0,C 180,E1 -14705.757,E2 -14705.757} C_VEL
LIN {X 0,Y 360.382,Z 351.045,A -85,B 0,C 180,E1 -14708.316,E2 -14708.316} C_VEL
LIN {X 0,Y 352.358,Z 335.012,A -85,B 0,C 180,E1 -14709.778,E2 -14709.778} C_VEL
LIN {X 0,Y 345.181,Z 322.576,A -85,B 0,C 180,E1 -14711.12,E2 -14711.12} C_VEL
LIN {X 0,Y 334.923,Z 307.086,A -85,B 0,C 180,E1 -14713.126,E2 -14713.126} C_VEL
LIN {X 0,Y 331.638,Z 302.515,A -85,B 0,C 180,E1 -14713.798,E2 -14713.798} C_VEL
LIN {X 0,Y 329.664,Z 299.331,A -85,B 0,C 180,E1 -14714.225,E2 -14714.225} C_VEL
LIN {X 0,Y 327.25,Z 296.478,A -85,B 0,C 180,E1 -14714.727,E2 -14714.727} C_VEL
LIN {X 0,Y 326.54,Z 294.113,A -85,B 0,C 180,E1 -14714.938,E2 -14714.938} C_VEL
LIN {X 0,Y 326.574,Z 294.109,A -85,B 0,C 180,E1 -14718.154,E2 -14718.154} C_VEL
LIN {X 0,Y 326.622,Z 294.11,A -85,B 0,C 180,E1 -14721.391,E2 -14721.391} C_VEL
LIN {X 0,Y 326.618,Z 294.112,A -85,B 0,C 180,E1 -14724.851,E2 -14724.851} C_VEL
LIN {X 0,Y 326.606,Z 294.096,A -85,B 0,C 180,E1 -14727.455,E2 -14727.455} C_VEL
LIN {X 0,Y 326.646,Z 294.109,A -85,B 0,C 180,E1 -14730.339,E2 -14730.339} C_VEL
LIN {X 0,Y 326.688,Z 294.102,A -85,B 0,C 180,E1 -14734.516,E2 -14734.516} C_VEL
LIN {X 0,Y 326.644,Z 294.085,A -85,B 0,C 180,E1 -14738.545,E2 -14738.545} C_VEL
LIN {X 0,Y 326.743,Z 294.097,A -85,B 0,C 180,E1 -14741.177,E2 -14741.177} C_VEL
LIN {X 0,Y 326.761,Z 294.077,A -85,B 0,C 180,E1 -14745.433,E2 -14745.433} C_VEL
LIN {X 0,Y 326.767,Z 294.078,A -85,B 0,C 180,E1 -14748.839,E2 -14748.839} C_VEL
LIN {X 0,Y 326.977,Z 294.06,A -85,B 0,C 180,E1 -14752.59,E2 -14752.59} C_VEL
LIN {X 0,Y 326.775,Z 294.084,A -85,B 0,C 180,E1 -14755.065,E2 -14755.065} C_VEL
LIN {X 0,Y 327.043,Z 294.03,A -85,B 0,C 180,E1 -14757.537,E2 -14757.537} C_VEL
LIN {X 0,Y 327.196,Z 294.039,A -85,B 0,C 180,E1 -14760,E2 -14760} C_VEL
LIN {X 0,Y 327.045,Z 294.041,A -85,B 0,C 180,E1 -14762.463,E2 -14762.463} C_VEL
LIN {X 0,Y 326.994,Z 294.06,A -85,B 0,C 180,E1 -14766.169,E2 -14766.169} C_VEL
LIN {X 0,Y 326.912,Z 294.066,A -85,B 0,C 180,E1 -14768.655,E2 -14768.655} C_VEL
LIN {X 0,Y 326.732,Z 294.09,A -85,B 0,C 180,E1 -14772.421,E2 -14772.421} C_VEL
LIN {X 0,Y 326.752,Z 294.092,A -85,B 0,C 180,E1 -14774.957,E2 -14774.957} C_VEL
LIN {X 0,Y 326.731,Z 294.095,A -85,B 0,C 180,E1 -14778.838,E2 -14778.838} C_VEL
LIN {X 0,Y 326.618,Z 294.116,A -85,B 0,C 180,E1 -14782.787,E2 -14782.787} C_VEL
LIN {X 0,Y 326.688,Z 294.109,A -85,B 0,C 180,E1 -14785.484,E2 -14785.484} C_VEL
LIN {X 0,Y 326.658,Z 294.109,A -85,B 0,C 180,E1 -14789.659,E2 -14789.659} C_VEL
LIN {X 0,Y 326.604,Z 294.12,A -85,B 0,C 180,E1 -14794.019,E2 -14794.019} C_VEL
LIN {X 0,Y 326.625,Z 294.118,A -85,B 0,C 180,E1 -14797.239,E2 -14797.239} C_VEL
LIN {X 0,Y 326.575,Z 294.124,A -85,B 0,C 180,E1 -14801.131,E2 -14801.131} C_VEL
LIN {X 0,Y 326.563,Z 294.171,A -85,B 0,C 180,E1 -14803.032,E2 -14803.032} C_VEL
LIN {X 0,Y 330.644,Z 304.519,A -85,B 0,C 180,E1 -14805.729,E2 -14805.729} C_VEL
LIN {X 0,Y 340.415,Z 320.419,A -85,B 0,C 180,E1 -14807.746,E2 -14807.746} C_VEL
LIN {X 0,Y 348.667,Z 335.337,A -85,B 0,C 180,E1 -14809.355,E2 -14809.355} C_VEL
LIN {X 0,Y 355.908,Z 349.551,A -85,B 0,C 180,E1 -14810.705,E2 -14810.705} C_VEL
LIN {X 0,Y 360.218,Z 358.746,A -85,B 0,C 180,E1 -14811.489,E2 -14811.489} C_VEL
LIN {X 0,Y 354.553,Z 512.855,A -85,B 0,C 180,E1 -14814.639,E2 -14814.639} C_VEL
LIN {X 0,Y 353.116,Z 529.736,A -85,B 0,C 180,E1 -14815.183,E2 -14815.183} C_VEL
LIN {X 0,Y 351.223,Z 545.93,A -85,B 0,C 180,E1 -14815.925,E2 -14815.925} C_VEL
LIN {X 0,Y 349.009,Z 561.786,A -85,B 0,C 180,E1 -14816.893,E2 -14816.893} C_VEL
LIN {X 0,Y 346.561,Z 576.421,A -85,B 0,C 180,E1 -14818.009,E2 -14818.009} C_VEL
LIN {X 0,Y 343.727,Z 591.455,A -85,B 0,C 180,E1 -14819.429,E2 -14819.429} C_VEL
LIN {X 0,Y 340.756,Z 605.191,A -85,B 0,C 180,E1 -14821.009,E2 -14821.009} C_VEL
LIN {X 0,Y 337.928,Z 617.932,A -85,B 0,C 180,E1 -14822.772,E2 -14822.772} C_VEL
LIN {X 0,Y 335.388,Z 629.342,A -85,B 0,C 180,E1 -14824.642,E2 -14824.642} C_VEL
LIN {X 0,Y 332.884,Z 639.91,A -85,B 0,C 180,E1 -14826.681,E2 -14826.681} C_VEL
LIN {X 0,Y 330.497,Z 650.295,A -85,B 0,C 180,E1 -14829.074,E2 -14829.074} C_VEL
LIN {X 0,Y 328.581,Z 659.445,A -85,B 0,C 180,E1 -14831.61,E2 -14831.61} C_VEL
LIN {X 0,Y 327.216,Z 666.093,A -85,B 0,C 180,E1 -14833.787,E2 -14833.787} C_VEL
LIN {X 0,Y 325.975,Z 673.794,A -85,B 0,C 180,E1 -14836.916,E2 -14836.916} C_VEL
LIN {X 0,Y 325.189,Z 679.657,A -85,B 0,C 180,E1 -14840.044,E2 -14840.044} C_VEL
LIN {X 0,Y 324.943,Z 683.091,A -85,B 0,C 180,E1 -14842.544,E2 -14842.544} C_VEL
LIN {X 0,Y 324.851,Z 685.589,A -85,B 0,C 180,E1 -14845.036,E2 -14845.036} C_VEL
LIN {X 0,Y 324.825,Z 686.998,A -85,B 0,C 180,E1 -14847.52,E2 -14847.52} C_VEL
LIN {X 0,Y 324.871,Z 687.529,A -85,B 0,C 180,E1 -14850,E2 -14850} C_VEL
LIN {X 0,Y 324.825,Z 686.992,A -85,B 0,C 180,E1 -14852.48,E2 -14852.48} C_VEL
LIN {X 0,Y 324.851,Z 685.576,A -85,B 0,C 180,E1 -14854.964,E2 -14854.964} C_VEL
LIN {X 0,Y 324.943,Z 683.074,A -85,B 0,C 180,E1 -14857.456,E2 -14857.456} C_VEL
LIN {X 0,Y 325.189,Z 679.635,A -85,B 0,C 180,E1 -14859.956,E2 -14859.956} C_VEL
LIN {X 0,Y 325.966,Z 673.764,A -85,B 0,C 180,E1 -14863.084,E2 -14863.084} C_VEL
LIN {X 0,Y 327.215,Z 666.049,A -85,B 0,C 180,E1 -14866.213,E2 -14866.213} C_VEL
LIN {X 0,Y 328.99,Z 657.355,A -85,B 0,C 180,E1 -14869.012,E2 -14869.012} C_VEL
LIN {X 0,Y 330.989,Z 647.976,A -85,B 0,C 180,E1 -14871.486,E2 -14871.486} C_VEL
LIN {X 0,Y 333.244,Z 638.335,A -85,B 0,C 180,E1 -14873.622,E2 -14873.622} C_VEL
LIN {X 0,Y 335.827,Z 627.167,A -85,B 0,C 180,E1 -14875.726,E2 -14875.726} C_VEL
LIN {X 0,Y 338.594,Z 614.877,A -85,B 0,C 180,E1 -14877.673,E2 -14877.673} C_VEL
LIN {X 0,Y 341.481,Z 601.518,A -85,B 0,C 180,E1 -14879.43,E2 -14879.43} C_VEL
LIN {X 0,Y 344.357,Z 587.63,A -85,B 0,C 180,E1 -14880.943,E2 -14880.943} C_VEL
LIN {X 0,Y 347.137,Z 572.771,A -85,B 0,C 180,E1 -14882.274,E2 -14882.274} C_VEL
LIN {X 0,Y 349.618,Z 557.445,A -85,B 0,C 180,E1 -14883.387,E2 -14883.387} C_VEL
LIN {X 0,Y 351.697,Z 541.706,A -85,B 0,C 180,E1 -14884.282,E2 -14884.282} C_VEL
LIN {X 0,Y 353.447,Z 525.623,A -85,B 0,C 180,E1 -14884.953,E2 -14884.953} C_VEL
LIN {X 0,Y 354.718,Z 509.456,A -85,B 0,C 180,E1 -14885.42,E2 -14885.42} C_VEL
LIN {X 0,Y 360.129,Z 358.62,A -85,B 0,C 180,E1 -14888.502,E2 -14888.502} C_VEL
LIN {X 0,Y 351.141,Z 339.997,A -85,B 0,C 180,E1 -14890.154,E2 -14890.154} C_VEL
LIN {X 0,Y 341.442,Z 322.221,A -85,B 0,C 180,E1 -14892.019,E2 -14892.019} C_VEL
LIN {X 0,Y 332.63,Z 307.691,A -85,B 0,C 180,E1 -14893.813,E2 -14893.813} C_VEL
LIN {X 0,Y 330.414,Z 303.992,A -85,B 0,C 180,E1 -14894.319,E2 -14894.319} C_VEL
LIN {X 0,Y 326.562,Z 294.115,A -85,B 0,C 180,E1 -14896.967,E2 -14896.967} C_VEL
LIN {X 0,Y 326.609,Z 294.105,A -85,B 0,C 180,E1 -14900.773,E2 -14900.773} C_VEL
LIN {X 0,Y 326.61,Z 294.107,A -85,B 0,C 180,E1 -14904.48,E2 -14904.48} C_VEL
LIN {X 0,Y 326.605,Z 294.107,A -85,B 0,C 180,E1 -14907.456,E2 -14907.456} C_VEL
LIN {X 0,Y 326.658,Z 294.102,A -85,B 0,C 180,E1 -14910.341,E2 -14910.341} C_VEL
LIN {X 0,Y 326.688,Z 294.105,A -85,B 0,C 180,E1 -14914.516,E2 -14914.516} C_VEL
LIN {X 0,Y 326.644,Z 294.092,A -85,B 0,C 180,E1 -14918.545,E2 -14918.545} C_VEL
LIN {X 0,Y 326.743,Z 294.075,A -85,B 0,C 180,E1 -14921.178,E2 -14921.178} C_VEL
LIN {X 0,Y 326.761,Z 294.069,A -85,B 0,C 180,E1 -14925.433,E2 -14925.433} C_VEL
LIN {X 0,Y 326.768,Z 294.087,A -85,B 0,C 180,E1 -14928.839,E2 -14928.839} C_VEL
LIN {X 0,Y 326.957,Z 294.041,A -85,B 0,C 180,E1 -14932.59,E2 -14932.59} C_VEL
LIN {X 0,Y 326.988,Z 294.032,A -85,B 0,C 180,E1 -14933.831,E2 -14933.831} C_VEL
LIN {X 0,Y 327.046,Z 294.058,A -85,B 0,C 180,E1 -14937.537,E2 -14937.537} C_VEL
LIN {X 0,Y 327.177,Z 294.011,A -85,B 0,C 180,E1 -14940,E2 -14940} C_VEL
LIN {X 0,Y 327.044,Z 294.04,A -85,B 0,C 180,E1 -14942.463,E2 -14942.463} C_VEL
LIN {X 0,Y 326.96,Z 294.047,A -85,B 0,C 180,E1 -14946.589,E2 -14946.589} C_VEL
LIN {X 0,Y 326.804,Z 294.071,A -85,B 0,C 180,E1 -14949.907,E2 -14949.907} C_VEL
LIN {X 0,Y 326.758,Z 294.077,A -85,B 0,C 180,E1 -14953.686,E2 -14953.686} C_VEL
LIN {X 0,Y 326.698,Z 294.095,A -85,B 0,C 180,E1 -14957.528,E2 -14957.528} C_VEL
LIN {X 0,Y 326.657,Z 294.094,A -85,B 0,C 180,E1 -14960.135,E2 -14960.135} C_VEL
LIN {X 0,Y 326.65,Z 294.105,A -85,B 0,C 180,E1 -14964.129,E2 -14964.129} C_VEL
LIN {X 0,Y 326.681,Z 294.083,A -85,B 0,C 180,E1 -14966.858,E2 -14966.858} C_VEL
LIN {X 0,Y 326.638,Z 294.111,A -85,B 0,C 180,E1 -14970.612,E2 -14970.612} C_VEL
LIN {X 0,Y 326.606,Z 294.11,A -85,B 0,C 180,E1 -14974.02,E2 -14974.02} C_VEL
LIN {X 0,Y 326.626,Z 294.092,A -85,B 0,C 180,E1 -14977.239,E2 -14977.239} C_VEL
LIN {X 0,Y 326.577,Z 294.106,A -85,B 0,C 180,E1 -14981.131,E2 -14981.131} C_VEL
LIN {X 0,Y 326.537,Z 294.114,A -85,B 0,C 180,E1 -14984.948,E2 -14984.948} C_VEL
LIN {X 0,Y 326.559,Z 294.299,A -85,B 0,C 180,E1 -14985.213,E2 -14985.213} C_VEL
LIN {X 0,Y 327.535,Z 296.964,A -85,B 0,C 180,E1 -14985.464,E2 -14985.464} C_VEL
LIN {X 0,Y 329.761,Z 299.505,A -85,B 0,C 180,E1 -14985.923,E2 -14985.923} C_VEL
LIN {X 0,Y 331.886,Z 302.797,A -85,B 0,C 180,E1 -14986.376,E2 -14986.376} C_VEL
LIN {X 0,Y 333.315,Z 304.868,A -85,B 0,C 180,E1 -14986.672,E2 -14986.672} C_VEL
LIN {X 0,Y 341.285,Z 316.601,A -85,B 0,C 180,E1 -14988.258,E2 -14988.258} C_VEL
LIN {X 0,Y 349.103,Z 329.099,A -85,B 0,C 180,E1 -14989.734,E2 -14989.734} C_VEL
LIN {X 0,Y 356.753,Z 343.624,A -85,B 0,C 180,E1 -14991.145,E2 -14991.145} C_VEL
LIN {X 0,Y 360.304,Z 350.851,A -85,B 0,C 180,E1 -14991.782,E2 -14991.782} C_VEL
LIN {X 0,Y 355.081,Z 494.276,A -85,B 0,C 180,E1 -14994.717,E2 -14994.717} C_VEL
LIN {X 0,Y 353.87,Z 510.475,A -85,B 0,C 180,E1 -14995.225,E2 -14995.225} C_VEL
LIN {X 0,Y 352.254,Z 526.623,A -85,B 0,C 180,E1 -14995.952,E2 -14995.952} C_VEL
LIN {X 0,Y 350.278,Z 541.937,A -85,B 0,C 180,E1 -14996.856,E2 -14996.856} C_VEL
LIN {X 0,Y 347.891,Z 557.245,A -85,B 0,C 180,E1 -14998.009,E2 -14998.009} C_VEL
LIN {X 0,Y 345.256,Z 572.166,A -85,B 0,C 180,E1 -14999.41,E2 -14999.41} C_VEL
LIN {X 0,Y 342.667,Z 584.957,A -85,B 0,C 180,E1 -15000.85,E2 -15000.85} C_VEL
LIN {X 0,Y 339.788,Z 598.027,A -85,B 0,C 180,E1 -15002.6,E2 -15002.6} C_VEL
LIN {X 0,Y 336.837,Z 610.891,A -85,B 0,C 180,E1 -15004.677,E2 -15004.677} C_VEL
LIN {X 0,Y 334.204,Z 621.736,A -85,B 0,C 180,E1 -15006.778,E2 -15006.778} C_VEL
LIN {X 0,Y 332.032,Z 631,A -85,B 0,C 180,E1 -15008.91,E2 -15008.91} C_VEL
LIN {X 0,Y 329.892,Z 640.016,A -85,B 0,C 180,E1 -15011.364,E2 -15011.364} C_VEL
LIN {X 0,Y 328.229,Z 647.544,A -85,B 0,C 180,E1 -15013.838,E2 -15013.838} C_VEL
LIN {X 0,Y 326.732,Z 655.103,A -85,B 0,C 180,E1 -15016.947,E2 -15016.947} C_VEL
LIN {X 0,Y 325.733,Z 660.84,A -85,B 0,C 180,E1 -15020.061,E2 -15020.061} C_VEL
LIN {X 0,Y 325.293,Z 664.197,A -85,B 0,C 180,E1 -15022.552,E2 -15022.552} C_VEL
LIN {X 0,Y 325.05,Z 666.636,A -85,B 0,C 180,E1 -15025.039,E2 -15025.039} C_VEL
LIN {X 0,Y 324.89,Z 668.023,A -85,B 0,C 180,E1 -15027.52,E2 -15027.52} C_VEL
LIN {X 0,Y 324.877,Z 668.556,A -85,B 0,C 180,E1 -15030,E2 -15030} C_VEL
LIN {X 0,Y 324.889,Z 668.064,A -85,B 0,C 180,E1 -15032.48,E2 -15032.48} C_VEL
LIN {X 0,Y 325.05,Z 666.717,A -85,B 0,C 180,E1 -15034.961,E2 -15034.961} C_VEL
LIN {X 0,Y 325.291,Z 664.319,A -85,B 0,C 180,E1 -15037.448,E2 -15037.448} C_VEL
LIN {X 0,Y 325.725,Z 661.011,A -85,B 0,C 180,E1 -15039.94,E2 -15039.94} C_VEL
LIN {X 0,Y 326.694,Z 655.325,A -85,B 0,C 180,E1 -15043.055,E2 -15043.055} C_VEL
LIN {X 0,Y 328.209,Z 647.838,A -85,B 0,C 180,E1 -15046.163,E2 -15046.163} C_VEL
LIN {X 0,Y 330.089,Z 639.351,A -85,B 0,C 180,E1 -15048.947,E2 -15048.947} C_VEL
LIN {X 0,Y 331.959,Z 631.406,A -85,B 0,C 180,E1 -15051.095,E2 -15051.095} C_VEL
LIN {X 0,Y 334.498,Z 620.748,A -85,B 0,C 180,E1 -15053.528,E2 -15053.528} C_VEL
LIN {X 0,Y 337.133,Z 609.739,A -85,B 0,C 180,E1 -15055.63,E2 -15055.63} C_VEL
LIN {X 0,Y 340.187,Z 596.702,A -85,B 0,C 180,E1 -15057.699,E2 -15057.699} C_VEL
LIN {X 0,Y 342.089,Z 587.998,A -85,B 0,C 180,E1 -15058.876,E2 -15058.876} C_VEL
LIN {X 0,Y 342.417,Z 583.496,A -85,B 0,C 180,E1 -15059.5,E2 -15059.5} C_VEL
LIN {X 0,Y 340.492,Z 568.465,A -85,B 0,C 180,E1 -15061.657,E2 -15061.657} C_VEL
LIN {X 0,Y 340.825,Z 563.473,A -85,B 0,C 180,E1 -15062.193,E2 -15062.193} C_VEL
LIN {X 0,Y 343.329,Z 549.364,A -85,B 0,C 180,E1 -15063.376,E2 -15063.376} C_VEL
LIN {X 0,Y 345.527,Z 534.683,A -85,B 0,C 180,E1 -15064.363,E2 -15064.363} C_VEL
LIN {X 0,Y 347.354,Z 518.648,A -85,B 0,C 180,E1 -15065.214,E2 -15065.214} C_VEL
LIN {X 0,Y 348.896,Z 502.256,A -85,B 0,C 180,E1 -15065.834,E2 -15065.834} C_VEL
LIN {X 0,Y 349.802,Z 484.468,A -85,B 0,C 180,E1 -15066.294,E2 -15066.294} C_VEL
LIN {X 0,Y 354.756,Z 353.435,A -85,B 0,C 180,E1 -15068.981,E2 -15068.981} C_VEL
LIN {X 0,Y 346.964,Z 337.881,A -85,B 0,C 180,E1 -15070.452,E2 -15070.452} C_VEL
LIN {X 0,Y 340.659,Z 327.015,A -85,B 0,C 180,E1 -15071.669,E2 -15071.669} C_VEL
LIN {X 0,Y 330.828,Z 312.051,A -85,B 0,C 180,E1 -15073.652,E2 -15073.652} C_VEL
LIN {X 0,Y 325.123,Z 303.979,A -85,B 0,C 180,E1 -15074.872,E2 -15074.872} C_VEL
LIN {X 0,Y 322.861,Z 300.65,A -85,B 0,C 180,E1 -15075.379,E2 -15075.379} C_VEL
LIN {X 0,Y 321.804,Z 299.382,A -85,B 0,C 180,E1 -15075.611,E2 -15075.611} C_VEL
LIN {X 0,Y 320.061,Z 297.032,A -85,B 0,C 180,E1 -15076.007,E2 -15076.007} C_VEL
LIN {X 0,Y 319.514,Z 294.988,A -85,B 0,C 180,E1 -15076.214,E2 -15076.214} C_VEL
LIN {X 0,Y 319.557,Z 294.988,A -85,B 0,C 180,E1 -15080.331,E2 -15080.331} C_VEL
LIN {X 0,Y 319.578,Z 294.987,A -85,B 0,C 180,E1 -15084.457,E2 -15084.457} C_VEL
LIN {X 0,Y 319.529,Z 294.98,A -85,B 0,C 180,E1 -15088.138,E2 -15088.138} C_VEL
LIN {X 0,Y 319.609,Z 294.966,A -85,B 0,C 180,E1 -15091.59,E2 -15091.59} C_VEL
LIN {X 0,Y 319.604,Z 294.987,A -85,B 0,C 180,E1 -15095.304,E2 -15095.304} C_VEL
LIN {X 0,Y 319.595,Z 294.961,A -85,B 0,C 180,E1 -15098.047,E2 -15098.047} C_VEL
LIN {X 0,Y 319.687,Z 294.978,A -85,B 0,C 180,E1 -15100.962,E2 -15100.962} C_VEL
LIN {X 0,Y 319.729,Z 294.95,A -85,B 0,C 180,E1 -15105.276,E2 -15105.276} C_VEL
LIN {X 0,Y 319.755,Z 294.938,A -85,B 0,C 180,E1 -15109.873,E2 -15109.873} C_VEL
LIN {X 0,Y 319.931,Z 294.937,A -85,B 0,C 180,E1 -15112.426,E2 -15112.426} C_VEL
LIN {X 0,Y 319.745,Z 294.961,A -85,B 0,C 180,E1 -15114.956,E2 -15114.956} C_VEL
LIN {X 0,Y 319.987,Z 294.908,A -85,B 0,C 180,E1 -15117.482,E2 -15117.482} C_VEL
LIN {X 0,Y 320.148,Z 294.917,A -85,B 0,C 180,E1 -15120,E2 -15120} C_VEL
LIN {X 0,Y 319.988,Z 294.918,A -85,B 0,C 180,E1 -15122.517,E2 -15122.517} C_VEL
LIN {X 0,Y 319.95,Z 294.938,A -85,B 0,C 180,E1 -15126.305,E2 -15126.305} C_VEL
LIN {X 0,Y 319.84,Z 294.943,A -85,B 0,C 180,E1 -15128.848,E2 -15128.848} C_VEL
LIN {X 0,Y 319.679,Z 294.97,A -85,B 0,C 180,E1 -15132.7,E2 -15132.7} C_VEL
LIN {X 0,Y 319.697,Z 294.97,A -85,B 0,C 180,E1 -15135.295,E2 -15135.295} C_VEL
LIN {X 0,Y 319.672,Z 294.978,A -85,B 0,C 180,E1 -15139.255,E2 -15139.255} C_VEL
LIN {X 0,Y 319.568,Z 294.993,A -85,B 0,C 180,E1 -15143.319,E2 -15143.319} C_VEL
LIN {X 0,Y 319.632,Z 294.987,A -85,B 0,C 180,E1 -15146.088,E2 -15146.088} C_VEL
LIN {X 0,Y 319.587,Z 294.995,A -85,B 0,C 180,E1 -15148.934,E2 -15148.934} C_VEL
LIN {X 0,Y 319.53,Z 295.002,A -85,B 0,C 180,E1 -15151.862,E2 -15151.862} C_VEL
LIN {X 0,Y 319.577,Z 294.99,A -85,B 0,C 180,E1 -15155.543,E2 -15155.543} C_VEL
LIN {X 0,Y 319.555,Z 294.999,A -85,B 0,C 180,E1 -15158.01,E2 -15158.01} C_VEL
LIN {X 0,Y 319.53,Z 295.033,A -85,B 0,C 180,E1 -15161.91,E2 -15161.91} C_VEL
LIN {X 0,Y 323.178,Z 304.24,A -85,B 0,C 180,E1 -15164.424,E2 -15164.424} C_VEL
LIN {X 0,Y 333.128,Z 320.033,A -85,B 0,C 180,E1 -15166.593,E2 -15166.593} C_VEL
LIN {X 0,Y 341.062,Z 333.941,A -85,B 0,C 180,E1 -15168.218,E2 -15168.218} C_VEL
LIN {X 0,Y 349.834,Z 350.873,A -85,B 0,C 180,E1 -15169.926,E2 -15169.926} C_VEL
LIN {X 0,Y 354.584,Z 361.06,A -85,B 0,C 180,E1 -15170.825,E2 -15170.825} C_VEL
LIN {X 0,Y 350.024,Z 480.802,A -85,B 0,C 180,E1 -15173.276,E2 -15173.276} C_VEL
LIN {X 0,Y 348.729,Z 513.317,A -85,B 0,C 180,E1 -15173.979,E2 -15173.979} C_VEL
LIN {X 0,Y 347.22,Z 530.457,A -85,B 0,C 180,E1 -15174.548,E2 -15174.548} C_VEL
LIN {X 0,Y 345.347,Z 545.729,A -85,B 0,C 180,E1 -15175.263,E2 -15175.263} C_VEL
LIN {X 0,Y 343.064,Z 561.584,A -85,B 0,C 180,E1 -15176.243,E2 -15176.243} C_VEL
LIN {X 0,Y 340.522,Z 576.217,A -85,B 0,C 180,E1 -15177.372,E2 -15177.372} C_VEL
LIN {X 0,Y 337.588,Z 591.25,A -85,B 0,C 180,E1 -15178.812,E2 -15178.812} C_VEL
LIN {X 0,Y 334.481,Z 604.984,A -85,B 0,C 180,E1 -15180.411,E2 -15180.411} C_VEL
LIN {X 0,Y 331.548,Z 617.724,A -85,B 0,C 180,E1 -15182.203,E2 -15182.203} C_VEL
LIN {X 0,Y 328.826,Z 629.465,A -85,B 0,C 180,E1 -15184.167,E2 -15184.167} C_VEL
LIN {X 0,Y 325.934,Z 641.148,A -85,B 0,C 180,E1 -15186.49,E2 -15186.49} C_VEL
LIN {X 0,Y 323.517,Z 651.218,A -85,B 0,C 180,E1 -15188.904,E2 -15188.904} C_VEL
LIN {X 0,Y 321.507,Z 660.254,A -85,B 0,C 180,E1 -15191.521,E2 -15191.521} C_VEL
LIN {X 0,Y 319.981,Z 667.535,A -85,B 0,C 180,E1 -15194.065,E2 -15194.065} C_VEL
LIN {X 0,Y 318.982,Z 673.585,A -85,B 0,C 180,E1 -15196.624,E2 -15196.624} C_VEL
LIN {X 0,Y 318.114,Z 679.448,A -85,B 0,C 180,E1 -15199.82,E2 -15199.82} C_VEL
LIN {X 0,Y 317.859,Z 682.883,A -85,B 0,C 180,E1 -15202.377,E2 -15202.377} C_VEL
LIN {X 0,Y 317.769,Z 685.382,A -85,B 0,C 180,E1 -15204.925,E2 -15204.925} C_VEL
LIN {X 0,Y 317.746,Z 686.792,A -85,B 0,C 180,E1 -15207.465,E2 -15207.465} C_VEL
LIN {X 0,Y 317.779,Z 687.321,A -85,B 0,C 180,E1 -15210,E2 -15210} C_VEL
LIN {X 0,Y 317.746,Z 686.785,A -85,B 0,C 180,E1 -15212.535,E2 -15212.535} C_VEL
LIN {X 0,Y 317.769,Z 685.368,A -85,B 0,C 180,E1 -15215.075,E2 -15215.075} C_VEL
LIN {X 0,Y 317.859,Z 682.865,A -85,B 0,C 180,E1 -15217.623,E2 -15217.623} C_VEL
LIN {X 0,Y 318.114,Z 679.425,A -85,B 0,C 180,E1 -15220.18,E2 -15220.18} C_VEL
LIN {X 0,Y 318.972,Z 673.553,A -85,B 0,C 180,E1 -15223.376,E2 -15223.376} C_VEL
LIN {X 0,Y 319.98,Z 667.493,A -85,B 0,C 180,E1 -15225.935,E2 -15225.935} C_VEL
LIN {X 0,Y 321.512,Z 660.199,A -85,B 0,C 180,E1 -15228.479,E2 -15228.479} C_VEL
LIN {X 0,Y 323.477,Z 651.316,A -85,B 0,C 180,E1 -15231.054,E2 -15231.054} C_VEL
LIN {X 0,Y 325.958,Z 641.074,A -85,B 0,C 180,E1 -15233.508,E2 -15233.508} C_VEL
LIN {X 0,Y 328.767,Z 629.481,A -85,B 0,C 180,E1 -15235.815,E2 -15235.815} C_VEL
LIN {X 0,Y 331.537,Z 617.607,A -85,B 0,C 180,E1 -15237.798,E2 -15237.798} C_VEL
LIN {X 0,Y 334.486,Z 604.843,A -85,B 0,C 180,E1 -15239.588,E2 -15239.588} C_VEL
LIN {X 0,Y 337.509,Z 591.073,A -85,B 0,C 180,E1 -15241.196,E2 -15241.196} C_VEL
LIN {X 0,Y 340.51,Z 576.014,A -85,B 0,C 180,E1 -15242.63,E2 -15242.63} C_VEL
LIN {X 0,Y 343.046,Z 561.325,A -85,B 0,C 180,E1 -15243.759,E2 -15243.759} C_VEL
LIN {X 0,Y 345.339,Z 545.398,A -85,B 0,C 180,E1 -15244.738,E2 -15244.738} C_VEL
LIN {X 0,Y 347.177,Z 529.991,A -85,B 0,C 180,E1 -15245.457,E2 -15245.457} C_VEL
LIN {X 0,Y 348.72,Z 513.667,A -85,B 0,C 180,E1 -15245.985,E2 -15245.985} C_VEL
LIN {X 0,Y 350.451,Z 467.344,A -85,B 0,C 180,E1 -15246.986,E2 -15246.986} C_VEL
LIN {X 0,Y 354.512,Z 361.839,A -85,B 0,C 180,E1 -15249.14,E2 -15249.14} C_VEL
LIN {X 0,Y 354.178,Z 360.312,A -85,B 0,C 180,E1 -15249.222,E2 -15249.222} C_VEL
LIN {X 0,Y 345.987,Z 343.307,A -85,B 0,C 180,E1 -15250.783,E2 -15250.783} C_VEL
LIN {X 0,Y 336.47,Z 325.759,A -85,B 0,C 180,E1 -15252.68,E2 -15252.68} C_VEL
LIN {X 0,Y 328.029,Z 311.8,A -85,B 0,C 180,E1 -15254.46,E2 -15254.46} C_VEL
LIN {X 0,Y 322.932,Z 303.622,A -85,B 0,C 180,E1 -15255.642,E2 -15255.642} C_VEL
LIN {X 0,Y 319.531,Z 294.987,A -85,B 0,C 180,E1 -15258.09,E2 -15258.09} C_VEL
LIN {X 0,Y 319.555,Z 294.985,A -85,B 0,C 180,E1 -15261.99,E2 -15261.99} C_VEL
LIN {X 0,Y 319.557,Z 294.984,A -85,B 0,C 180,E1 -15265.123,E2 -15265.123} C_VEL
LIN {X 0,Y 319.568,Z 294.989,A -85,B 0,C 180,E1 -15269.058,E2 -15269.058} C_VEL
LIN {X 0,Y 319.606,Z 294.981,A -85,B 0,C 180,E1 -15272.498,E2 -15272.498} C_VEL
LIN {X 0,Y 319.603,Z 294.982,A -85,B 0,C 180,E1 -15275.304,E2 -15275.304} C_VEL
LIN {X 0,Y 319.595,Z 294.98,A -85,B 0,C 180,E1 -15278.048,E2 -15278.048} C_VEL
LIN {X 0,Y 319.687,Z 294.95,A -85,B 0,C 180,E1 -15280.962,E2 -15280.962} C_VEL
LIN {X 0,Y 319.729,Z 294.946,A -85,B 0,C 180,E1 -15285.276,E2 -15285.276} C_VEL
LIN {X 0,Y 319.751,Z 294.968,A -85,B 0,C 180,E1 -15289.873,E2 -15289.873} C_VEL
LIN {X 0,Y 319.911,Z 294.919,A -85,B 0,C 180,E1 -15292.426,E2 -15292.426} C_VEL
LIN {X 0,Y 319.744,Z 294.945,A -85,B 0,C 180,E1 -15294.956,E2 -15294.956} C_VEL
LIN {X 0,Y 319.99,Z 294.937,A -85,B 0,C 180,E1 -15297.483,E2 -15297.483} C_VEL
LIN {X 0,Y 320.129,Z 294.888,A -85,B 0,C 180,E1 -15300,E2 -15300} C_VEL
LIN {X 0,Y 319.988,Z 294.919,A -85,B 0,C 180,E1 -15302.518,E2 -15302.518} C_VEL
LIN {X 0,Y 319.922,Z 294.923,A -85,B 0,C 180,E1 -15306.576,E2 -15306.576} C_VEL
LIN {X 0,Y 319.751,Z 294.953,A -85,B 0,C 180,E1 -15310.128,E2 -15310.128} C_VEL
LIN {X 0,Y 319.729,Z 294.938,A -85,B 0,C 180,E1 -15314.724,E2 -15314.724} C_VEL
LIN {X 0,Y 319.687,Z 294.975,A -85,B 0,C 180,E1 -15319.038,E2 -15319.038} C_VEL
LIN {X 0,Y 319.562,Z 294.972,A -85,B 0,C 180,E1 -15323.32,E2 -15323.32} C_VEL
LIN {X 0,Y 319.633,Z 294.973,A -85,B 0,C 180,E1 -15326.088,E2 -15326.088} C_VEL
LIN {X 0,Y 319.587,Z 294.967,A -85,B 0,C 180,E1 -15328.934,E2 -15328.934} C_VEL
LIN {X 0,Y 319.531,Z 294.989,A -85,B 0,C 180,E1 -15331.862,E2 -15331.862} C_VEL
LIN {X 0,Y 319.579,Z 294.988,A -85,B 0,C 180,E1 -15335.543,E2 -15335.543} C_VEL
LIN {X 0,Y 319.558,Z 294.983,A -85,B 0,C 180,E1 -15339.669,E2 -15339.669} C_VEL
LIN {X 0,Y 319.52,Z 294.99,A -85,B 0,C 180,E1 -15343.7,E2 -15343.7} C_VEL
LIN {X 0,Y 319.509,Z 295.1,A -85,B 0,C 180,E1 -15343.959,E2 -15343.959} C_VEL
LIN {X 0,Y 320.466,Z 297.818,A -85,B 0,C 180,E1 -15344.224,E2 -15344.224} C_VEL
LIN {X 0,Y 322.801,Z 300.539,A -85,B 0,C 180,E1 -15344.736,E2 -15344.736} C_VEL
LIN {X 0,Y 325.117,Z 303.962,A -85,B 0,C 180,E1 -15345.255,E2 -15345.255} C_VEL
LIN {X 0,Y 326.293,Z 305.597,A -85,B 0,C 180,E1 -15345.51,E2 -15345.51} C_VEL
LIN {X 0,Y 334.779,Z 317.937,A -85,B 0,C 180,E1 -15347.286,E2 -15347.286} C_VEL
LIN {X 0,Y 344.209,Z 332.886,A -85,B 0,C 180,E1 -15349.137,E2 -15349.137} C_VEL
LIN {X 0,Y 351.724,Z 347.24,A -85,B 0,C 180,E1 -15350.57,E2 -15350.57} C_VEL
LIN {X 0,Y 354.65,Z 353.145,A -85,B 0,C 180,E1 -15351.112,E2 -15351.112} C_VEL
LIN {X 0,Y 349.368,Z 493.965,A -85,B 0,C 180,E1 -15354.035,E2 -15354.035} C_VEL
LIN {X 0,Y 348.073,Z 510.695,A -85,B 0,C 180,E1 -15354.559,E2 -15354.559} C_VEL
LIN {X 0,Y 346.409,Z 526.838,A -85,B 0,C 180,E1 -15355.296,E2 -15355.296} C_VEL
LIN {X 0,Y 344.36,Z 542.151,A -85,B 0,C 180,E1 -15356.211,E2 -15356.211} C_VEL
LIN {X 0,Y 341.887,Z 557.458,A -85,B 0,C 180,E1 -15357.379,E2 -15357.379} C_VEL
LIN {X 0,Y 339.408,Z 571.106,A -85,B 0,C 180,E1 -15358.669,E2 -15358.669} C_VEL
LIN {X 0,Y 336.742,Z 584.002,A -85,B 0,C 180,E1 -15360.114,E2 -15360.114} C_VEL
LIN {X 0,Y 333.716,Z 597.265,A -85,B 0,C 180,E1 -15361.887,E2 -15361.887} C_VEL
LIN {X 0,Y 330.797,Z 609.366,A -85,B 0,C 180,E1 -15363.842,E2 -15363.842} C_VEL
LIN {X 0,Y 328.004,Z 620.474,A -85,B 0,C 180,E1 -15365.977,E2 -15365.977} C_VEL
LIN {X 0,Y 325.672,Z 629.885,A -85,B 0,C 180,E1 -15368.116,E2 -15368.116} C_VEL
LIN {X 0,Y 323.367,Z 639.223,A -85,B 0,C 180,E1 -15370.644,E2 -15370.644} C_VEL
LIN {X 0,Y 321.345,Z 647.755,A -85,B 0,C 180,E1 -15373.482,E2 -15373.482} C_VEL
LIN {X 0,Y 319.755,Z 655.313,A -85,B 0,C 180,E1 -15376.657,E2 -15376.657} C_VEL
LIN {X 0,Y 318.711,Z 661.049,A -85,B 0,C 180,E1 -15379.839,E2 -15379.839} C_VEL
LIN {X 0,Y 318.221,Z 664.406,A -85,B 0,C 180,E1 -15382.385,E2 -15382.385} C_VEL
LIN {X 0,Y 317.961,Z 666.845,A -85,B 0,C 180,E1 -15384.928,E2 -15384.928} C_VEL
LIN {X 0,Y 317.811,Z 668.23,A -85,B 0,C 180,E1 -15387.465,E2 -15387.465} C_VEL
LIN {X 0,Y 317.785,Z 668.763,A -85,B 0,C 180,E1 -15390,E2 -15390} C_VEL
LIN {X 0,Y 317.81,Z 668.27,A -85,B 0,C 180,E1 -15392.535,E2 -15392.535} C_VEL
LIN {X 0,Y 317.961,Z 666.925,A -85,B 0,C 180,E1 -15395.072,E2 -15395.072} C_VEL
LIN {X 0,Y 318.218,Z 664.526,A -85,B 0,C 180,E1 -15397.615,E2 -15397.615} C_VEL
LIN {X 0,Y 318.704,Z 661.218,A -85,B 0,C 180,E1 -15400.161,E2 -15400.161} C_VEL
LIN {X 0,Y 319.722,Z 655.533,A -85,B 0,C 180,E1 -15403.344,E2 -15403.344} C_VEL
LIN {X 0,Y 321.312,Z 648.046,A -85,B 0,C 180,E1 -15406.52,E2 -15406.52} C_VEL
LIN {X 0,Y 323.325,Z 639.558,A -85,B 0,C 180,E1 -15409.359,E2 -15409.359} C_VEL
LIN {X 0,Y 325.484,Z 630.636,A -85,B 0,C 180,E1 -15411.802,E2 -15411.802} C_VEL
LIN {X 0,Y 327.953,Z 620.955,A -85,B 0,C 180,E1 -15414.027,E2 -15414.027} C_VEL
LIN {X 0,Y 330.687,Z 609.945,A -85,B 0,C 180,E1 -15416.167,E2 -15416.167} C_VEL
LIN {X 0,Y 333.403,Z 598.869,A -85,B 0,C 180,E1 -15417.97,E2 -15417.97} C_VEL
LIN {X 0,Y 336.291,Z 585.927,A -85,B 0,C 180,E1 -15419.758,E2 -15419.758} C_VEL
LIN {X 0,Y 339.258,Z 572.156,A -85,B 0,C 180,E1 -15421.33,E2 -15421.33} C_VEL
LIN {X 0,Y 340.825,Z 563.473,A -85,B 0,C 180,E1 -15422.193,E2 -15422.193} C_VEL
LIN {X 0,Y 341.2,Z 558.441,A -85,B 0,C 180,E1 -15422.711,E2 -15422.711} C_VEL
LIN {X 0,Y 339.284,Z 542.78,A -85,B 0,C 180,E1 -15424.439,E2 -15424.439} C_VEL
LIN {X 0,Y 339.449,Z 536.57,A -85,B 0,C 180,E1 -15424.931,E2 -15424.931} C_VEL
LIN {X 0,Y 341.378,Z 520.367,A -85,B 0,C 180,E1 -15425.834,E2 -15425.834} C_VEL
LIN {X 0,Y 343.002,Z 504.761,A -85,B 0,C 180,E1 -15426.455,E2 -15426.455} C_VEL
LIN {X 0,Y 344.04,Z 487.14,A -85,B 0,C 180,E1 -15426.938,E2 -15426.938} C_VEL
LIN {X 0,Y 349.204,Z 355.886,A -85,B 0,C 180,E1 -15429.663,E2 -15429.663} C_VEL
LIN {X 0,Y 342.173,Z 341.833,A -85,B 0,C 180,E1 -15431.036,E2 -15431.036} C_VEL
LIN {X 0,Y 336.189,Z 331.482,A -85,B 0,C 180,E1 -15432.228,E2 -15432.228} C_VEL
LIN {X 0,Y 326.9,Z 317.213,A -85,B 0,C 180,E1 -15434.161,E2 -15434.161} C_VEL
LIN {X 0,Y 320.976,Z 308.837,A -85,B 0,C 180,E1 -15435.466,E2 -15435.466} C_VEL
LIN {X 0,Y 318.263,Z 305,A -85,B 0,C 180,E1 -15436.09,E2 -15436.09} C_VEL
LIN {X 0,Y 316.022,Z 301.759,A -85,B 0,C 180,E1 -15436.622,E2 -15436.622} C_VEL
LIN {X 0,Y 315.224,Z 300.607,A -85,B 0,C 180,E1 -15436.814,E2 -15436.814} C_VEL
LIN {X 0,Y 313.298,Z 298.374,A -85,B 0,C 180,E1 -15437.267,E2 -15437.267} C_VEL
LIN {X 0,Y 312.479,Z 295.873,A -85,B 0,C 180,E1 -15437.539,E2 -15437.539} C_VEL
LIN {X 0,Y 312.501,Z 295.873,A -85,B 0,C 180,E1 -15440.971,E2 -15440.971} C_VEL
LIN {X 0,Y 312.531,Z 295.86,A -85,B 0,C 180,E1 -15444.22,E2 -15444.22} C_VEL
LIN {X 0,Y 312.502,Z 295.852,A -85,B 0,C 180,E1 -15447.333,E2 -15447.333} C_VEL
LIN {X 0,Y 312.542,Z 295.85,A -85,B 0,C 180,E1 -15451.279,E2 -15451.279} C_VEL
LIN {X 0,Y 312.584,Z 295.86,A -85,B 0,C 180,E1 -15454.711,E2 -15454.711} C_VEL
LIN {X 0,Y 312.586,Z 295.834,A -85,B 0,C 180,E1 -15457.529,E2 -15457.529} C_VEL
LIN {X 0,Y 312.636,Z 295.851,A -85,B 0,C 180,E1 -15461.656,E2 -15461.656} C_VEL
LIN {X 0,Y 312.692,Z 295.833,A -85,B 0,C 180,E1 -15465.686,E2 -15465.686} C_VEL
LIN {X 0,Y 312.7,Z 295.818,A -85,B 0,C 180,E1 -15469.642,E2 -15469.642} C_VEL
LIN {X 0,Y 312.87,Z 295.812,A -85,B 0,C 180,E1 -15472.254,E2 -15472.254} C_VEL
LIN {X 0,Y 312.715,Z 295.838,A -85,B 0,C 180,E1 -15474.842,E2 -15474.842} C_VEL
LIN {X 0,Y 312.988,Z 295.792,A -85,B 0,C 180,E1 -15478.713,E2 -15478.713} C_VEL
LIN {X 0,Y 312.988,Z 295.807,A -85,B 0,C 180,E1 -15481.286,E2 -15481.286} C_VEL
LIN {X 0,Y 312.714,Z 295.819,A -85,B 0,C 180,E1 -15485.157,E2 -15485.157} C_VEL
LIN {X 0,Y 312.87,Z 295.824,A -85,B 0,C 180,E1 -15487.746,E2 -15487.746} C_VEL
LIN {X 0,Y 312.667,Z 295.828,A -85,B 0,C 180,E1 -15491.671,E2 -15491.671} C_VEL
LIN {X 0,Y 312.697,Z 295.842,A -85,B 0,C 180,E1 -15494.887,E2 -15494.887} C_VEL
LIN {X 0,Y 312.628,Z 295.855,A -85,B 0,C 180,E1 -15499.236,E2 -15499.236} C_VEL
LIN {X 0,Y 312.544,Z 295.87,A -85,B 0,C 180,E1 -15502.789,E2 -15502.789} C_VEL
LIN {X 0,Y 312.6,Z 295.863,A -85,B 0,C 180,E1 -15505.936,E2 -15505.936} C_VEL
LIN {X 0,Y 312.543,Z 295.867,A -85,B 0,C 180,E1 -15509.65,E2 -15509.65} C_VEL
LIN {X 0,Y 312.517,Z 295.873,A -85,B 0,C 180,E1 -15513.689,E2 -15513.689} C_VEL
LIN {X 0,Y 312.523,Z 295.875,A -85,B 0,C 180,E1 -15517.385,E2 -15517.385} C_VEL
LIN {X 0,Y 312.487,Z 295.895,A -85,B 0,C 180,E1 -15520.709,E2 -15520.709} C_VEL
LIN {X 0,Y 313.032,Z 297.869,A -85,B 0,C 180,E1 -15521.259,E2 -15521.259} C_VEL
LIN {X 0,Y 315.513,Z 303.672,A -85,B 0,C 180,E1 -15522.976,E2 -15522.976} C_VEL
LIN {X 0,Y 325.603,Z 319.237,A -85,B 0,C 180,E1 -15525.311,E2 -15525.311} C_VEL
LIN {X 0,Y 333.653,Z 332.947,A -85,B 0,C 180,E1 -15527.049,E2 -15527.049} C_VEL
LIN {X 0,Y 343.143,Z 351.049,A -85,B 0,C 180,E1 -15528.991,E2 -15528.991} C_VEL
LIN {X 0,Y 349.014,Z 363.632,A -85,B 0,C 180,E1 -15530.148,E2 -15530.148} C_VEL
LIN {X 0,Y 343.084,Z 512.215,A -85,B 0,C 180,E1 -15533.259,E2 -15533.259} C_VEL
LIN {X 0,Y 341.53,Z 529.342,A -85,B 0,C 180,E1 -15533.82,E2 -15533.82} C_VEL
LIN {X 0,Y 339.709,Z 544.227,A -85,B 0,C 180,E1 -15534.51,E2 -15534.51} C_VEL
LIN {X 0,Y 337.505,Z 559.391,A -85,B 0,C 180,E1 -15535.429,E2 -15535.429} C_VEL
LIN {X 0,Y 334.859,Z 574.354,A -85,B 0,C 180,E1 -15536.569,E2 -15536.569} C_VEL
LIN {X 0,Y 331.801,Z 589.616,A -85,B 0,C 180,E1 -15538.026,E2 -15538.026} C_VEL
LIN {X 0,Y 328.55,Z 603.6,A -85,B 0,C 180,E1 -15539.645,E2 -15539.645} C_VEL
LIN {X 0,Y 325.737,Z 615.557,A -85,B 0,C 180,E1 -15541.311,E2 -15541.311} C_VEL
LIN {X 0,Y 322.994,Z 626.685,A -85,B 0,C 180,E1 -15543.14,E2 -15543.14} C_VEL
LIN {X 0,Y 320.04,Z 637.997,A -85,B 0,C 180,E1 -15545.34,E2 -15545.34} C_VEL
LIN {X 0,Y 317.287,Z 648.864,A -85,B 0,C 180,E1 -15547.88,E2 -15547.88} C_VEL
LIN {X 0,Y 315.128,Z 658.008,A -85,B 0,C 180,E1 -15550.456,E2 -15550.456} C_VEL
LIN {X 0,Y 313.41,Z 665.675,A -85,B 0,C 180,E1 -15553.051,E2 -15553.051} C_VEL
LIN {X 0,Y 311.998,Z 673.376,A -85,B 0,C 180,E1 -15556.319,E2 -15556.319} C_VEL
LIN {X 0,Y 311.051,Z 679.24,A -85,B 0,C 180,E1 -15559.586,E2 -15559.586} C_VEL
LIN {X 0,Y 310.774,Z 682.675,A -85,B 0,C 180,E1 -15562.202,E2 -15562.202} C_VEL
LIN {X 0,Y 310.682,Z 685.174,A -85,B 0,C 180,E1 -15564.809,E2 -15564.809} C_VEL
LIN {X 0,Y 310.669,Z 686.585,A -85,B 0,C 180,E1 -15567.407,E2 -15567.407} C_VEL
LIN {X 0,Y 310.689,Z 687.115,A -85,B 0,C 180,E1 -15570,E2 -15570} C_VEL
LIN {X 0,Y 310.669,Z 686.578,A -85,B 0,C 180,E1 -15572.593,E2 -15572.593} C_VEL
LIN {X 0,Y 310.721,Z 684.795,A -85,B 0,C 180,E1 -15575.616,E2 -15575.616} C_VEL
LIN {X 0,Y 310.774,Z 682.656,A -85,B 0,C 180,E1 -15577.798,E2 -15577.798} C_VEL
LIN {X 0,Y 311.051,Z 679.215,A -85,B 0,C 180,E1 -15580.414,E2 -15580.414} C_VEL
LIN {X 0,Y 311.986,Z 673.342,A -85,B 0,C 180,E1 -15583.682,E2 -15583.682} C_VEL
LIN {X 0,Y 313.409,Z 665.625,A -85,B 0,C 180,E1 -15586.949,E2 -15586.949} C_VEL
LIN {X 0,Y 315.388,Z 656.931,A -85,B 0,C 180,E1 -15589.866,E2 -15589.866} C_VEL
LIN {X 0,Y 317.619,Z 647.552,A -85,B 0,C 180,E1 -15592.438,E2 -15592.438} C_VEL
LIN {X 0,Y 320.076,Z 637.91,A -85,B 0,C 180,E1 -15594.657,E2 -15594.657} C_VEL
LIN {X 0,Y 322.808,Z 626.993,A -85,B 0,C 180,E1 -15596.795,E2 -15596.795} C_VEL
LIN {X 0,Y 325.981,Z 614.453,A -85,B 0,C 180,E1 -15598.842,E2 -15598.842} C_VEL
LIN {X 0,Y 329.083,Z 601.093,A -85,B 0,C 180,E1 -15600.656,E2 -15600.656} C_VEL
LIN {X 0,Y 332.254,Z 586.852,A -85,B 0,C 180,E1 -15602.247,E2 -15602.247} C_VEL
LIN {X 0,Y 335.129,Z 572.343,A -85,B 0,C 180,E1 -15603.58,E2 -15603.58} C_VEL
LIN {X 0,Y 337.824,Z 557.016,A -85,B 0,C 180,E1 -15604.715,E2 -15604.715} C_VEL
LIN {X 0,Y 340.041,Z 541.276,A -85,B 0,C 180,E1 -15605.632,E2 -15605.632} C_VEL
LIN {X 0,Y 341.913,Z 525.187,A -85,B 0,C 180,E1 -15606.316,E2 -15606.316} C_VEL
LIN {X 0,Y 343.244,Z 508.984,A -85,B 0,C 180,E1 -15606.794,E2 -15606.794} C_VEL
LIN {X 0,Y 348.908,Z 363.233,A -85,B 0,C 180,E1 -15609.85,E2 -15609.85} C_VEL
LIN {X 0,Y 340.07,Z 345.011,A -85,B 0,C 180,E1 -15611.595,E2 -15611.595} C_VEL
LIN {X 0,Y 330.896,Z 328.148,A -85,B 0,C 180,E1 -15613.5,E2 -15613.5} C_VEL
LIN {X 0,Y 321.807,Z 313.333,A -85,B 0,C 180,E1 -15615.501,E2 -15615.501} C_VEL
LIN {X 0,Y 317.086,Z 306.139,A -85,B 0,C 180,E1 -15616.6,E2 -15616.6} C_VEL
LIN {X 0,Y 315.333,Z 303.334,A -85,B 0,C 180,E1 -15617.067,E2 -15617.067} C_VEL
LIN {X 0,Y 313.847,Z 299.232,A -85,B 0,C 180,E1 -15618.235,E2 -15618.235} C_VEL
LIN {X 0,Y 312.536,Z 296.315,A -85,B 0,C 180,E1 -15619.14,E2 -15619.14} C_VEL
LIN {X 0,Y 312.488,Z 295.87,A -85,B 0,C 180,E1 -15619.291,E2 -15619.291} C_VEL
LIN {X 0,Y 312.523,Z 295.858,A -85,B 0,C 180,E1 -15622.615,E2 -15622.615} C_VEL
LIN {X 0,Y 312.517,Z 295.866,A -85,B 0,C 180,E1 -15626.311,E2 -15626.311} C_VEL
LIN {X 0,Y 312.543,Z 295.86,A -85,B 0,C 180,E1 -15630.35,E2 -15630.35} C_VEL
LIN {X 0,Y 312.601,Z 295.859,A -85,B 0,C 180,E1 -15634.064,E2 -15634.064} C_VEL
LIN {X 0,Y 312.585,Z 295.858,A -85,B 0,C 180,E1 -15637.529,E2 -15637.529} C_VEL
LIN {X 0,Y 312.636,Z 295.838,A -85,B 0,C 180,E1 -15641.657,E2 -15641.657} C_VEL
LIN {X 0,Y 312.692,Z 295.816,A -85,B 0,C 180,E1 -15645.686,E2 -15645.686} C_VEL
LIN {X 0,Y 312.696,Z 295.848,A -85,B 0,C 180,E1 -15649.642,E2 -15649.642} C_VEL
LIN {X 0,Y 312.851,Z 295.8,A -85,B 0,C 180,E1 -15652.254,E2 -15652.254} C_VEL
LIN {X 0,Y 312.714,Z 295.817,A -85,B 0,C 180,E1 -15654.843,E2 -15654.843} C_VEL
LIN {X 0,Y 312.987,Z 295.796,A -85,B 0,C 180,E1 -15658.714,E2 -15658.714} C_VEL
LIN {X 0,Y 312.987,Z 295.774,A -85,B 0,C 180,E1 -15661.287,E2 -15661.287} C_VEL
LIN {X 0,Y 312.715,Z 295.842,A -85,B 0,C 180,E1 -15665.158,E2 -15665.158} C_VEL
LIN {X 0,Y 312.852,Z 295.789,A -85,B 0,C 180,E1 -15667.746,E2 -15667.746} C_VEL
LIN {X 0,Y 312.668,Z 295.85,A -85,B 0,C 180,E1 -15671.672,E2 -15671.672} C_VEL
LIN {X 0,Y 312.699,Z 295.812,A -85,B 0,C 180,E1 -15674.888,E2 -15674.888} C_VEL
LIN {X 0,Y 312.628,Z 295.853,A -85,B 0,C 180,E1 -15679.236,E2 -15679.236} C_VEL
LIN {X 0,Y 312.528,Z 295.84,A -85,B 0,C 180,E1 -15682.782,E2 -15682.782} C_VEL
LIN {X 0,Y 312.601,Z 295.852,A -85,B 0,C 180,E1 -15685.936,E2 -15685.936} C_VEL
LIN {X 0,Y 312.544,Z 295.856,A -85,B 0,C 180,E1 -15689.65,E2 -15689.65} C_VEL
LIN {X 0,Y 312.518,Z 295.867,A -85,B 0,C 180,E1 -15693.689,E2 -15693.689} C_VEL
LIN {X 0,Y 312.519,Z 295.847,A -85,B 0,C 180,E1 -15697.386,E2 -15697.386} C_VEL
LIN {X 0,Y 312.489,Z 295.866,A -85,B 0,C 180,E1 -15700.709,E2 -15700.709} C_VEL
LIN {X 0,Y 312.49,Z 295.879,A -85,B 0,C 180,E1 -15702.623,E2 -15702.623} C_VEL
